(* CODESYS project UPMRACING_Driverless.project

Project tree, tasks and I/O mapping:
  Device : HY-TTC 580, TTControl, order no. n/a, version 1.2.0.0
    application Application
      libraries: Standard, * (System); lib500, 1.2.0.0 (TTControl); lib500_types, 1.2.0.0 (TTControl); lib500_syscom, 1.2.0.0 (TTControl); lib500_can2, 0.2.0.5 (TTControl); Util, * (System); Base Control Library Unsafe, 0.4.0.2 (TTControl)
      task MainTask (cyclic, interval t#10ms, priority 3, watchdog t#1000ms x 1) calls PLC_PRG
      task _ErrorCallback (externalevent, external event ErrorCallback, priority 1) calls _ErrorCB_PRG
      task _NotificationCallback (externalevent, external event NotificationCallback, priority 0) calls _NotificationCB_PRG
      program PLC_PRG [ST]
      program _NotificationCB_PRG [ST]
      program _ErrorCB_PRG [ST]
      global variables GVL
      program cl_split_byte [ST]
      CAN_Rx/
        function block CAN0_RX_Inverters [ST]
        function block CAN1_RX_V_0 [ST]
        function block CAN2_RX_V_0 [ST]
        function block CAN3_RX_V_0 [ST]
      CAN_Tx/
        function block CAN0_TX_Inverters [ST]
        function block CAN1_TX_V_0 [ST]
        function block CAN2_TX_V_0 [ST]
        function block CAN2_TX_V_1 [ST]
      UPM03/
        function block CAN_TX_V_1_4 [ST]
        function block CAN_RX_V_1_2 [ST]
        function block UPMRacing_14E_StateMachine_Antigua [ST]
      V_1/
        function block UPMRacing_14E_StateMachine [ST]
        global variables GVL_CONSTS
        function block UPMRacing_14E_StateMachine_vieja [ST]
        function block PLC_CODER_TIMER [ST]
    CANs : CANs, TTControl, order no. n/a, version 1.2.0.0
      CAN0 : CAN0, TTControl, order no. n/a, version 1.2.0.0
      CAN1 : CAN1, TTControl, order no. n/a, version 1.2.0.0
      CAN2 : CAN2, TTControl, order no. n/a, version 1.2.0.0
          settings: Baudrate = 1000
      CAN3 : CAN3, TTControl, order no. n/a, version 1.2.0.0
      CAN4 : CAN4, TTControl, order no. n/a, version 1.2.0.0
      CAN5 : CAN5, TTControl, order no. n/a, version 1.2.0.0
      CAN6 : CAN6, TTControl, order no. n/a, version 1.2.0.0
          settings: Baudrate = 250
    System : System, TTControl, order no. n/a, version 1.2.0.0
        output Application.GVL.PowerStage : BYTE  // mode
        output Application.GVL.gSafetySwitch0 : BYTE  // mode
        output Application.GVL.gSensorSupply : BYTE  // mode
        output Application.GVL.gSensorSupply : BYTE  // mode
        output Application.GVL.gSensorSupply_10 : BYTE  // mode
        output Application.GVL.Shutdown : BIT  // shutdown
        input  Application.GVL.K15 : DWORD  // Terminal_15.value
        input  Application.GVL.Wake_Up : DWORD  // WakeUp.value
        unmapped channels: error, error, mode, error, mode, error, error, error, error, error, enable_error_group_0, enable_error_group_1, enable_error_group_2, diag_status, safe_state, error, driver_init_error, UBAT, Terminal_15, WakeUp, Temperature, SSW0, SSW1, SSW2, SSUP0, SSUP1, SSUP2, status, write, boot_error, trigger_error, Powerstage, SSW0, SSW1, SSW2, SSUP0, SSUP1, SSUP2, Terminal_15, WakeUp,
          ExtShutOff0, ExtShutOff1, ExtShutOff2
      Analog_Inputs_2Mode_10V : AIN_2Mode_10V, TTControl, order no. n/a, version 1.2.0.0
        Pin 107
          <Vacío>
        Pin 131
          <Vacío>
        Pin 108
          LV_Cell_2 : IoDrvADC2Mode10, TTControl, order no. n/a, version 1.2.0.0
              input  Application.GVL.LV_Cell_2 : lib500_types.IO_ADC_STATUS  // status
              unmapped channels: reset_trigger, reset_count, reset_error
        Pin 132
          <Vacío>
        Pin 109
          LV_Cell_1 : IoDrvADC2Mode10, TTControl, order no. n/a, version 1.2.0.0
              input  Application.GVL.LV_Cell_1 : lib500_types.IO_ADC_STATUS  // status
              unmapped channels: reset_trigger, reset_count, reset_error
        Pin 133
          <Empty>
        Pin 110
          <Vacío>
        Pin 134
          <Empty>
      Analog_Inputs_2Mode_32V : AIN_2Mode_32V, TTControl, order no. n/a, version 1.2.0.0
        Pin 111
          Drive_Button : IoDrvADC2Mode32, TTControl, order no. n/a, version 1.2.0.0
              input  Application.GVL.Drive_Button : lib500_types.IO_ADC_STATUS  // status
              unmapped channels: reset_trigger, reset_count, reset_error
        Pin 135
          Shutdown_Circuit : IoDrvADC2Mode32, TTControl, order no. n/a, version 1.2.0.0
              input  Application.GVL.Shutdown_Circuit : lib500_types.IO_ADC_STATUS  // status
              unmapped channels: reset_trigger, reset_count, reset_error
        Pin 112
          Reset_Button : IoDrvADC2Mode32, TTControl, order no. n/a, version 1.2.0.0
              input  Application.GVL.Reset_Button : lib500_types.IO_ADC_STATUS  // status
              unmapped channels: reset_trigger, reset_count, reset_error
        Pin 136
          LV_Cell_6 : IoDrvADC2Mode32, TTControl, order no. n/a, version 1.2.0.0
              input  Application.GVL.LV_Cell_6 : lib500_types.IO_ADC_STATUS  // status
              unmapped channels: reset_trigger, reset_count, reset_error
        Pin 113
          LV_Cell_8 : IoDrvADC2Mode32, TTControl, order no. n/a, version 1.2.0.0
              input  Application.GVL.LV_Cell_8 : lib500_types.IO_ADC_STATUS  // status
              unmapped channels: reset_trigger, reset_count, reset_error
        Pin 137
          LV_Cell_5 : IoDrvADC2Mode32, TTControl, order no. n/a, version 1.2.0.0
              input  Application.GVL.LV_Cell_5 : lib500_types.IO_ADC_STATUS  // status
              unmapped channels: reset_trigger, reset_count, reset_error
        Pin 114
          LV_Cell_7 : IoDrvADC2Mode32, TTControl, order no. n/a, version 1.2.0.0
              input  Application.GVL.LV_Cell_7 : lib500_types.IO_ADC_STATUS  // status
              unmapped channels: reset_trigger, reset_count, reset_error
        Pin 138
          LV_Cell_4 : IoDrvADC2Mode32, TTControl, order no. n/a, version 1.2.0.0
              input  Application.GVL.LV_Cell_4 : lib500_types.IO_ADC_STATUS  // status
              unmapped channels: reset_trigger, reset_count, reset_error
      Analog_Inputs_3Mode : AIN_3Mode, TTControl, order no. n/a, version 1.2.0.0
        Pin 103
          <Vacío>
        Pin 127
          <Empty>
        Pin 104
          <Empty>
        Pin 128
          <Empty>
        Pin 105
          <Empty>
        Pin 129
          <Empty>
        Pin 106
          <Empty>
        Pin 130
          <Empty>
      Digital_Outputs_HS : HSDOUT, TTControl, order no. n/a, version 1.2.0.0
        Pin 149
          Pre_Charge : IoDrvDOSafety, TTControl, order no. n/a, version 1.2.0.0
              output Application.GVL.Pre_Charge : BIT  // output
              unmapped channels: error_code, reset_trigger, reset_count, reset_error, current, voltage_feedback
        Pin 173
          RTDS : IoDrvDOSafety, TTControl, order no. n/a, version 1.2.0.0
              output Application.GVL.RTDS_Sound : BIT  // output
              unmapped channels: error_code, reset_trigger, reset_count, reset_error, current, voltage_feedback
        Pin 152
          Brake_Light : IoDrvDOSafety, TTControl, order no. n/a, version 1.2.0.0
              output Application.GVL.Brake_Light : BIT  // output
              unmapped channels: error_code, reset_trigger, reset_count, reset_error, current, voltage_feedback
        Pin 176
          <Vacío>
        Pin 155
          <Vacío>
        Pin 179
          <Vacío>
        Pin 158
          <Vacío>
        Pin 182
          <Vacío>
      Digital_Outputs_LS : LSDOUT, TTControl, order no. n/a, version 1.2.0.0
        Pin 251
          <Empty>
        Pin 238
          <Empty>
        Pin 252
          <Empty>
        Pin 239
          <Empty>
        Pin 253
          <Empty>
        Pin 240
          <Empty>
        Pin 254
          <Empty>
        Pin 241
          <Empty>
      PVG_Outputs : PVG, TTControl, order no. n/a, version 1.2.0.0
        Pin 161
          GVL_X15_EF2_INV_1_2 : IoDrvDODiag, TTControl, order no. n/a, version 1.2.0.0
              output Application.GVL.GVL_X15_EF2_INV_1_2 : BIT  // output
              input  Application.GVL.ERROR_GVL_X15_EF2_INV_1_2 : WORD  // error_code
              unmapped channels: reset_trigger, reset_count, reset_error, current, voltage_feedback
        Pin 185
          GVL_X15_EF2_INV_3_4 : IoDrvDODiag, TTControl, order no. n/a, version 1.2.0.0
              output Application.GVL.GVL_X15_EF2_INV_3_4 : BIT  // output
              input  Application.GVL.ERROR_GVL_X15_EF2_INV_3_4 : WORD  // error_code
              unmapped channels: reset_trigger, reset_count, reset_error, current, voltage_feedback
        Pin 188
          <Empty>
        Pin 164
          <Empty>
        Pin 191
          <Empty>
        Pin 167
          <Empty>
        Pin 194
          <Vacío>
        Pin 170
          <Empty>
      PWM_Outputs : PWM, TTControl, order no. n/a, version 1.2.0.0
        Safety_switch_0 : PWM_SSW0, TTControl, order no. n/a, version 1.2.0.0
          Pin 153
            <Vacío>
          Pin 177
            <Empty>
          Pin 156
            <Empty>
          Pin 180
            <Vacío>
          Pin 159
            <Empty>
          Pin 183
            <Empty>
          Pin 186
            <Empty>
          Pin 162
            <Empty>
          Pin 189
            <Empty>
          Pin 165
            <Empty>
          Pin 192
            <Empty>
          Pin 168
            <Empty>
          Pin 195
            <Empty>
          Pin 171
            <Empty>
        Safety_switch_1 : PWM_SSW1, TTControl, order no. n/a, version 1.2.0.0
          Pin 154
            <Empty>
          Pin 178
            <Empty>
          Pin 157
            <Empty>
          Pin 181
            <Empty>
          Pin 160
            <Empty>
          Pin 184
            <Empty>
          Pin 187
            <Empty>
          Pin 163
            <Empty>
          Pin 190
            <Empty>
          Pin 166
            <Empty>
          Pin 193
            <Empty>
          Pin 169
            <Empty>
          Pin 196
            <Vacío>
          Pin 172
            <Empty>
        Safety_switch_2 : PWM_SSW2, TTControl, order no. n/a, version 1.2.0.0
          Pin 101
            <Empty>
          Pin 125
            <Empty>
          Pin 150
            <Empty>
          Pin 174
            <Empty>
          Pin 102
            <Empty>
          Pin 126
            <Empty>
          Pin 151
            <Empty>
          Pin 175
            <Empty>
      Timer_Inputs_Cur : TIN_Cur, TTControl, order no. n/a, version 1.2.0.0
        Pin 115
          <Empty>
        Pin 139
          <Empty>
        Pin 116
          <Empty>
        Pin 140
          <Empty>
        Pin 117
          <Empty>
        Pin 141
          <Empty>
      Timer_Inputs : TIN, TTControl, order no. n/a, version 1.2.0.0
        Pin 122
          <Empty>
        Pin 146
          LV_Cell_3 : IoDrvADC, TTControl, order no. n/a, version 1.2.0.0
              input  Application.GVL.LV_Cell_3 : lib500_types.IO_ADC_STATUS  // status
        Pin 123
          <Empty>
        Pin 147
          <Empty>
        Pin 124
          <Empty>
        Pin 148
          <Empty>
*)

// Device/Application/GVL
(*24-04-2019 Se añade gSensorSupply para que la ECU alimente con 5V. También se añade g delante de gK15, porque sino no funciona. *)


{attribute 'qualified_only'}
VAR_GLOBAL
	
(*SYSTEM VARIABLES*)
	(*Para que funcione la alimentacion de los sensores*)
	(* Powerstage status variable *)
	PowerStage:lib500_types.IO_POWER_STATE:=lib500_types.IO_POWER_STATE.IO_POWER_OFF;	
	(* Sensor Supply status variable 5V*)
	gSensorSupply: lib500_types.IO_POWER_STATE := lib500_types.IO_POWER_STATE.IO_POWER_OFF;  
	(* Sensor Supply status variable 10V*)    
	gSensorSupply_10 	: lib500_types.IO_POWER_STATE := lib500_types.IO_POWER_STATE.IO_POWER_OFF;   
(*VARIABLES OUT PWM*)	
	gSafetySwitch0 	: lib500_types.IO_POWER_STATE := lib500_types.IO_POWER_STATE.IO_POWER_OFF;      (* Safey Switch 0 status variable *)  
	
	Shutdown	: BOOL 	:= FALSE;		(* Flag to shutdown controller by software *)
	K15		: DWORD := 0;			(* Voltage value of K15 pin *)
	Wake_Up	: DWORD := 0;			(* Voltage value of Wake_Up pin *)
	CALL_SAFE_SHUTDOWN:BOOL:=FALSE;
		
(*SENSORES ENTRADA ANALOGICA*)
	//AccPedal_1: lib500_types.IO_ADC_STATUS; (* Voltaje del potenciómetro *)
	//AccPedal_2: lib500_types.IO_ADC_STATUS;
	//Brake_Pedal: lib500_types.IO_ADC_STATUS;
	Reset_Button: lib500_types.IO_ADC_STATUS;
	Drive_Button: lib500_types.IO_ADC_STATUS;
	(*Steering_Wheel: lib500_types.IO_ADC_STATUS;*)
	Shutdown_Circuit: lib500_types.IO_ADC_STATUS;
	(*BMS LV*)
	LV_Cell_1: lib500_types.IO_ADC_STATUS;
	LV_Cell_2: lib500_types.IO_ADC_STATUS;
	LV_Cell_3: lib500_types.IO_ADC_STATUS;
	LV_Cell_4: lib500_types.IO_ADC_STATUS;
	LV_Cell_5: lib500_types.IO_ADC_STATUS;
	LV_Cell_6: lib500_types.IO_ADC_STATUS;
	LV_Cell_7: lib500_types.IO_ADC_STATUS;
	LV_Cell_8: lib500_types.IO_ADC_STATUS;
	LV_Cell_9: lib500_types.IO_ADC_STATUS;
	
		

	

(*CAN HANDLES*)

	(* Structure for sending  CAN messages *)
	H_CAN_TX_0:tCan;
	H_CAN_TX_1:tCan; 
	H_CAN_TX_2:tCan;
	H_CAN_TX_3:tCan;
	
	(* Structure for  receiving CAN messages *)
	H_CAN_RX_0:tCan; (* INV 1 & 2 & 3 & 4 *)
	H_CAN_RX_1:tCan;  (* AIM BMS Telemtry *)
	H_CAN_RX_2:tCan;  (* LVBMS Cooling FrontSups Telemetry *)
	H_CAN_RX_3:tCan;  (* DataLogger CTMD *)
	
(*DIGITAL_OUTPUTS*)
	Brake_Light: BOOL:=FALSE;
	Pre_Charge: BOOL:=FALSE; 
	RTDS_Sound: BOOL:=FALSE;

(*PWM VARIABLES*)	
	
	
	(*RTDS_Sound: WORD:=0;*)
	
	
(*GLOBAL VARIABLES*)	
	
	Estado: LREAL:=0;
	Estado_Error: LREAL:=0;
	Info_Inverter_Error: LREAL:=0; 
	
	(*ERRORS*)
		(* ERROR_GVL_X08_INV_1_2:lib500_types.IO_ERRORTYPE:=lib500_types.IO_errortype.IO_E_OK;
		ERROR_GVL_X08_INV_3_4:lib500_types.IO_ERRORTYPE:=lib500_types.IO_errortype.IO_E_OK;
		ERROR_GVL_X15_EF_INV_1_2:lib500_types.IO_ERRORTYPE:=lib500_types.IO_errortype.IO_E_OK;
		ERROR_GVL_X15_EF_INV_3_4:lib500_types.IO_ERRORTYPE:=lib500_types.IO_errortype.IO_E_OK;
		ERROR_GVL_X140_BE1_INV_1_2:lib500_types.IO_ERRORTYPE:=lib500_types.IO_errortype.IO_E_OK;
		ERROR_GVL_X140_BE1_INV_3_4:lib500_types.IO_ERRORTYPE:=lib500_types.IO_errortype.IO_E_OK;
		ERROR_GVL_X140_BE2_INV_1_2:lib500_types.IO_ERRORTYPE:=lib500_types.IO_errortype.IO_E_OK;
		ERROR_GVL_X140_BE2_INV_3_4:lib500_types.IO_ERRORTYPE:=lib500_types.IO_errortype.IO_E_OK;
		ERROR_GVL_X15_EF2_INV_1_2:lib500_types.IO_ERRORTYPE:=lib500_types.IO_errortype.IO_E_OK;
		ERROR_GVL_X15_EF2_INV_3_4:lib500_types.IO_ERRORTYPE:=lib500_types.IO_errortype.IO_E_OK; *)
END_VAR

// Device/Application/V_1/GVL_CONSTS
VAR_GLOBAL CONSTANT
	c_UPMRacing_14_IN_NO_ACTIVE: USINT := 0;
	c_UPMRacing_14E_StateMac_IN: USINT := 1;
	c_UPMRacing_14_IN_ERROR_PRE: USINT := 2;
	c_UPMRacing_14E_StateM_IN_L: USINT := 3;
	c_UPMRacing_14E_IN_POWER_MO: USINT := 4;
	c_UPMRacing_14E_StateMa_IN_: USINT := 5;
	c_UPMRa_IN_WAITING_FOR_INV_: USINT := 6;
	c_UPMRacing_14E_StateM_IN_W: USINT := 7;
	c_UPMRacing_14E_Sta_IN_Acce: USINT := 1;
	d_UPMRacing_14E_StateMac_IN: USINT := 2;
	c_UPM_IN_BRAKE_PLAUSIBILITY: USINT := 3;
	c_UPMRac_IN_IMPLAUSIBILITY_: USINT := 4;
	c_UPMRacing_14E_Stat_IN_PRE: USINT := 5;
	c_UPMRacing_14E_StateMach_I: USINT := 6;
	c_UPMRacing_14E_IN_PRE_CHAR: USINT := 1;
	c_UPMRacing_14E_IN_PRE_CHA: USINT := 2;
	c_UPMRacing_14E_St_IN_DRIVE: USINT := 1;
	d_UPMRacing_14E_StateMach_I: USINT := 2;
	c_UPMRacing_1_IN_POWER_FRON: USINT := 3;
	c_UPMR_IN_SHUTDOWN_SEQUENCE: USINT := 4;
	c_UPMRacing_14E_S_IN_HV_STA: USINT := 1;
	d_UPMRacing_14E_S_IN_HV_STA: USINT := 2;
	e_UPMRacing_14E_S_IN_HV_STA: USINT := 3;
	f_UPMRacing_14E_S_IN_HV_STA: USINT := 4;
	g_UPMRacing_14E_S_IN_HV_STA: USINT := 5;
	h_UPMRacing_14E_S_IN_HV_STA: USINT := 6;
	c_UPMRacing_14E_IN_INIT_PRE: USINT := 7;
	c_UPMRacing_14E_St_IN_INVER: USINT := 8;
	c_UPMRacing_14E_St_IN_HV_SH: USINT := 1;
	c_UPMRacing_14E_IN_INIT_DIS: USINT := 2;
	c_UPMRacing_14_IN_INIT_DISC: USINT := 3;
	c_IN_INVERTER_CONTROLLER_SH: USINT := 4;
	c_UPMRacing_14E_St_IN_ERROR: USINT := 2;
	c_UPMRacing_14E_St_IN_RESET: USINT := 3;
	c_UPMRacing_14E_Sta_IN_DRIV: USINT := 1;
	c_UPMRacing_14_IN_POWER_REA: USINT := 3;
	c_UPMRa_IN_SHUTDOWN_SEQUENC: USINT := 4;
	c_UPMRacing_14E_Sta_IN_RESE: USINT := 3;
	e_UPMRacing_14E_StateMac_IN: USINT := 1;
	c_UPMRacing_14E_State_IN_NO: USINT := 2;
	d_UPMRacing_14E_St_IN_RESET: USINT := 3;
	c_UPMRacing_14E_Stat_IN_LIG: USINT := 1;
	c_UPMRacing_14E_State_IN_LI: USINT := 2;
	SS_OUTPUT: SINT := 3;
	SS_INITIALIZE: SINT := 0;
	SS_STEP: SINT := 1;
END_VAR

// Device/Application/PLC_PRG
PROGRAM PLC_PRG
VAR
	InitPLC: BOOL := TRUE;		(* Initialization variable *)
	Counter: DWORD := 0;		(* Local counter *)
	UPMRacing_14E_StateMachine:UPMRacing_14E_StateMachine; 
	 
	Ignition_EVCU:LREAL:=0;
	ECU_ON_K15:REAL:=0;
	
	RTDS_Sound_PLC: UINT:=0;
END_VAR

(*FUNCIONES DE INICIO SEGURO CUANDO SE ENCIENDE LA ECU*)
	IF (InitPLC = TRUE) THEN
		(*FUNCIONES PARA INICIALIZAR CAN*)
			(*CAN_TX_0*)
				CanInit(	iEnable			:= TRUE,                                (* Initialiaze CAN *) 
								iChannel		:= 0, 									(* CAN Channel 1 *)
								iCAN			:= ADR(GVL.H_CAN_TX_0), 						(* Structure for sending / receiving CAN messages *)
								iBaudrate       := 500, 								(* 500 kBit *)
								iCanIdExtended  := FALSE, 								(* Standard CAN Frame *)
								iEcuCycleTime   := T#10MS);
			(*CAN_RX_0*)
				CanInit(	iEnable			:= TRUE,                                (* Initialiaze CAN *) 
								iChannel		:= 0, 									(* CAN Channel 1 *)
								iCAN			:= ADR(GVL.H_CAN_RX_0), 						(* Structure for sending / receiving CAN messages *)
								iBaudrate       :=500, 								(* 500 kBit *)
								iCanIdExtended  := FALSE, 								(* Standard CAN Frame *)
								iEcuCycleTime   := T#10MS);
		    (*CAN_TX_1*)					
			CanInit(	iEnable			:= TRUE,                                (* Initialiaze CAN *) 
								iChannel		:= 1, 									(* CAN Channel 1 *)
								iCAN			:= ADR(GVL.H_CAN_TX_1), 						(* Structure for sending / receiving CAN messages *)
								iBaudrate       := 500, 								(* 250 kBit *)
								iCanIdExtended  := FALSE, 								(* Standard CAN Frame *)
								iEcuCycleTime   := T#10MS);
			(*CAN_RX_1*)
				CanInit(	iEnable			:= TRUE,                                (* Initialiaze CAN *) 
								iChannel		:= 1, 									(* CAN Channel 1 *)
								iCAN			:= ADR(GVL.H_CAN_RX_1), 						(* Structure for sending / receiving CAN messages *)
								iBaudrate       := 500, 								(* 250 kBit *)
								iCanIdExtended  := FALSE, 								(* Standard CAN Frame *)
								iEcuCycleTime   := T#10MS); 
							
											
			(*CAN_TX_3*)					
			CanInit(	iEnable			:= TRUE,                                (* Initialiaze CAN *) 
								iChannel		:= 3, 									(* CAN Channel 1 *)
								iCAN			:= ADR(GVL.H_CAN_TX_3), 						(* Structure for sending / receiving CAN messages *)
								iBaudrate       := 500, 								(* 500 kBit *)
								iCanIdExtended  := FALSE, 								(* Standard CAN Frame *)
								iEcuCycleTime   := T#10MS);
			(*CAN_RX_3*)
				CanInit(	iEnable			:= TRUE,                                (* Initialiaze CAN *) 
								iChannel		:= 3, 									(* CAN Channel 1 *)
								iCAN			:= ADR(GVL.H_CAN_RX_3), 						(* Structure for sending / receiving CAN messages *)
								iBaudrate       := 500, 								(* 500 kBit *)
								iCanIdExtended  := FALSE, 								(* Standard CAN Frame *)
								iEcuCycleTime   := T#10MS);

						
		    (*CAN_TX_2*)					
			CanInit(	iEnable			:= TRUE,                                (* Initialiaze CAN *) 
								iChannel		:= 2, 									(* CAN Channel 1 *)
								iCAN			:= ADR(GVL.H_CAN_TX_2), 						(* Structure for sending / receiving CAN messages *)
								iBaudrate       := 500, 								(* 500 kBit *)
								iCanIdExtended  := FALSE, 								(* Standard CAN Frame *)
								iEcuCycleTime   := T#10MS);  
			(*CAN_RX_2*)
				CanInit(	iEnable			:= TRUE,                                (* Initialiaze CAN *) 
								iChannel		:= 2, 									(* CAN Channel 1 *)
								iCAN			:= ADR(GVL.H_CAN_RX_2), 						(* Structure for sending / receiving CAN messages *)
								iBaudrate       := 500, 								(* 500 kBit *)
								iCanIdExtended  := FALSE, 								(* Standard CAN Frame *)
								iEcuCycleTime   := T#10MS); 					
	    
        (*DIGITAL_OUTPUT_POWERSTAGE*)
		GVL.PowerStage:=lib500_types.IO_POWER_STATE.IO_POWER_ON;	
		
		(*INICIALIZAR SENSOR SUPPLY*)
		//GVL.gSensorSupply  := lib500_types.IO_POWER_STATE.IO_POWER_ON;		(* Switching on Sensor Supply 0 and 1 to get 5V for Potentiometers *)
		//GVL.gSensorSupply_10  := lib500_types.IO_POWER_STATE.IO_POWER_ON_10V;		(* Switching on Sensor Supply 2 to get 10V for other Purposes *)	
		
		(*INICIALIZAR PWM OUT*)
		//GVL.gSafetySwitch0 := lib500_types.IO_POWER_STATE.IO_POWER_ON;		(* Switching on Safety Switch for PWM use *)
		(*INICILIZAR MAQUINA DE ESTADOS*)	
			
		UPMRacing_14E_StateMachine(ssMethodType:=0);
		
		
		(*FIN INICIALIZACION*)
		InitPLC := FALSE;  
END_IF

(*DIGITAL INPUTS*)
	IF (gvl.K15>3000) THEN
		ECU_ON_K15:=1;
	END_IF

(*UPMRACING14E_STATE_MACHINE RUN*)
(*Es necesario igualar las variables gobales que vienen de entradas analogicas, al mismo tiempo que se asigna valor a las globales de salida*)
	UPMRacing_14E_StateMachine(ssMethodType:=1,
		
	
			 ); 
			
			(*GVL.RTDS_Sound:=UINT_TO_WORD(65535*RTDS_Sound_PLC/DWORD_TO_UINT(GVL.K15));*)
			
	
(*SHUTDOWN ECU*)
	IF (GVL.K15< 3000) THEN			(* K15 < 3V *)
		Counter := Counter + 1;			(* Increment counter cyclically *)
		IF (Counter >= 500) THEN		
			GVL.Shutdown := TRUE;  (* Shutdown controller only after 500 cycles *)	
		END_IF
	ELSE
		Counter := 0;					(* Reset counter if K15 is HIGH again *)
	END_IF

END_PROGRAM

// Device/Application/V_1/UPMRacing_14E_StateMachine
FUNCTION_BLOCK UPMRacing_14E_StateMachine
VAR_INPUT
	ssMethodType: SINT;
	MISSION_STATUS: USINT;
	SDC: BOOL;
	FRONT_AXLE_TRQ_REQUEST: UINT;
	REAR_AXLE_TRQ_REQUEST: UINT;
	STEER_REQUEST_deg: REAL;
	DIRECTION_REQUEST: BOOL;
	Accel_longitudinal_ms2: INT;
	Accel_lateral_ms2: INT;
	Yaw_rate_degps: INT;
	HANDSHAKE: BOOL;
	ESTOP_REQUEST: BOOL;
	LAP_COUNTER: USINT;
	CONES_COUNT_ACTUAL: USINT;
	CONES_COUNT_ALL: USINT;
	VEH_SPEED_ACTUAL: USINT;
	VEH_SPEED_DEMAND: USINT;
	FRONT_MOTOR_SPEED_MAX: UINT;
	REAR_MOTOR_SPEED_MAX: UINT;
	HYD_PRESS_F_REQ_pct: USINT;
	HYD_PRESS_R_REQ_pct: USINT;
END_VAR
VAR_OUTPUT
	State_ASSI: USINT;
	Steer_actual_deg: SINT;
	AI_ESTOP_REQUEST: BOOL;
	BMS_FAULT: BOOL;
	FR_WHEEL_SPEED: UINT;
	FL_WHEEL_SPEED: UINT;
	RR_WHEEL_SPEED: UINT;
	RL_WHEEL_SPEED: UINT;
	MISSION_STATUS_FAULT: BOOL;
	GO_SIGNAL: BOOL;
	AUTONOMOUS_BRAKING_FAULT: BOOL;
	BRAKE_PLAUSIBILITY_FAULT: BOOL;
	AI_COMMS_LOST_FAULT: BOOL;
	STATUS_EBS: USINT;
	TS_SWITCH_STATUS: BOOL;
	
			//FBTX_VCU2LOG_Dynamics1 
		Speed_actual_kmh: USINT;
		Speed_target_kmh: USINT;
		Steer_target_deg: SINT;
		Brake_actual_pct: USINT;
		Brake_target_pct: USINT;
		Drive_trq_actual_pct: SINT;
		Drive_trq_target_pct: SINT;
		
//FBTX_VCU2LOG_Status 		
		State_EBS: USINT; 
		AMI_STATE: USINT;
		State_steering: BOOL;
		State_service_brake: USINT;
		
//FBTX_VCU2AI_Status
		SHUTDOWN_REQUEST: BOOL;
		STEERING_STATUS: BOOL;
		AS_STATE: USINT;
		FAULT_STATUS: BOOL;
		WARNING_STATUS: BOOL;
		WARN_BATT_TEMP_HIGH: BOOL;
		WARN_BATT_SOC_LOW: BOOL;
		HVIL_OPEN_FAULT: BOOL;
		HVIL_SHORT_FAULT: BOOL;
		EBS_FAULT: BOOL;
		OFFBOARD_CHARGER_FAULT: BOOL;
		AI_COMMS_LOST: BOOL;
		CHARGE_PROCEDURE_FAULT: BOOL;
		SHUTDOWN_CAUSE: USINT;
		
		//FBTX_VCU2AI_Drive_F
		FRONT_AXLE_TRQ: INT;
		FRONT_AXLE_TRQ_MAX: UINT;
		
		//FBTX_VCU2AI_Drive_R
		REAR_AXLE_TRQ: INT;
		REAR_AXLE_TRQ_MAX: UINT;
		
				//FBTX_VCU2AI_Steer
		ANGLE: REAL;
		ANGLE_MAX: UINT;
		ANGLE_REQUEST: INT;
		
		//FBTX_VCU2AI_Brake 	
		HYD_PRESS_F_pct: USINT;
		HYD_PRESS_R_pct: USINT;
		STATUS_BRK: USINT;
		
		//FBTX_VCU2AI_Wheel_counts
		FL_PULSE_COUNT: UINT;
		FR_PULSE_COUNT: UINT;
		RL_PULSE_COUNT: UINT;
		RR_PULSE_COUNT: UINT;
		
		//VCU_STATUS
		SM_SYS: USINT;
		SM_AS: USINT;
		R1_AI2VCU_STATUS_TIMEOUT_ERROR: BOOL;
		R1_AI2VCU_DRIVE_F_TIMEOUT_ERROR: BOOL;
		R1_AI2VCU_DRIVE_R_TIMEOUT_ERROR: BOOL;
		R1_AI2VCU_STATUS_HANDSHAKE_ERROR: BOOL;
		R1_AI2VCU_STEER_TIMEOUT_ERROR: BOOL;
		R1_AI2VCU_BRAKE_TIMEOUT_ERROR: BOOL;
		SYS_ACTION_STATE: USINT;
		WARN_BRAKE_PLAUSIBILITY: BOOL;
		WARN_KL15_UNDER_V: BOOL;
		WARN_AI_ESTOP_REQ: BOOL;
		WARN_AI_COMMS_LOST: BOOL;
		WARN_AUTO_BRAKING: BOOL;
		WARN_MISSION_STATUS: BOOL;

		
		
END_VAR
VAR
	sf_internal_predicateOutput: BOOL;
	c_is_active_c3_UPMRacing_Dr: USINT;
	is_Main: USINT;
	temporalCounter_i1: PLC_CODER_TIMER;
	AS_SWITCH_STATUS: BOOL;
	//Llamadas a las funciones de CAN (Copiar)

	
//	CAN3_RX_V_0:CAN3_RX_V_0;	
	CAN2_RX_V_0:CAN2_RX_V_0;
	CAN1_RX_V_0:CAN1_RX_V_0;
	
	CAN2_TX_V_1:CAN2_TX_V_1;
	CAN1_TX_V_0:CAN1_TX_V_0;
	
END_VAR

CAN1_RX_V_0(
		
					Accel_longitudinal_ms2_CAN => Accel_longitudinal_ms2,
					Accel_lateral_ms2_CAN => Accel_lateral_ms2,
					Yaw_rate_degps_CAN => Yaw_rate_degps,
					HANDSHAKE_CAN => HANDSHAKE,
					ESTOP_REQUEST_CAN => ESTOP_REQUEST,
					MISSION_STATUS_CAN => MISSION_STATUS,
					DIRECTION_REQUEST_CAN => DIRECTION_REQUEST,
					LAP_COUNTER_CAN => LAP_COUNTER,
					CONES_COUNT_ACTUAL_CAN => CONES_COUNT_ACTUAL,
					CONES_COUNT_ALL_CAN => CONES_COUNT_ALL,
					VEH_SPEED_ACTUAL_CAN => VEH_SPEED_ACTUAL,
					VEH_SPEED_DEMAND_CAN => VEH_SPEED_DEMAND,
					FRONT_AXLE_TRQ_REQUEST_CAN => FRONT_AXLE_TRQ_REQUEST,
					FRONT_MOTOR_SPEED_MAX_CAN => FRONT_MOTOR_SPEED_MAX,
					REAR_AXLE_TRQ_REQUEST_CAN => REAR_AXLE_TRQ_REQUEST,
					REAR_MOTOR_SPEED_MAX_CAN => REAR_MOTOR_SPEED_MAX,
					STEER_REQUEST_deg_CAN => STEER_REQUEST_deg,
					HYD_PRESS_F_REQ_pct_CAN => HYD_PRESS_F_REQ_pct,
					HYD_PRESS_R_REQ_pct_CAN => HYD_PRESS_R_REQ_pct,

);
	(* *)
		 
CAN2_RX_V_0(
					ASMS_CAN => AS_SWITCH_STATUS,
					TSMS_CAN => TS_SWITCH_STATUS,
					GO_SIGNAL_CAN => GO_SIGNAL,
					SDC_CAN => SDC,
					MISSION_STATUS_FAULT_CAN => MISSION_STATUS_FAULT,
					AUTONOMOUS_BRAKING_FAULT_CAN => AUTONOMOUS_BRAKING_FAULT,
					COMMS_LOST_REQUEST_CAN => AI_COMMS_LOST_FAULT,
					BMS_FAULT_CAN => BMS_FAULT,
					EBS_Status_CAN => STATUS_EBS,
					FL_WHEEL_SPEED_CAN => FL_WHEEL_SPEED,
					FR_WHEEL_SPEED_CAN => FR_WHEEL_SPEED,
					RL_WHEEL_SPEED_CAN => RL_WHEEL_SPEED,
					RR_WHEEL_SPEED_CAN => RR_WHEEL_SPEED,
	
		);


CASE ssMethodType OF
    0: 
        (* SystemInitialize for Chart: '<Root>/UPMRacing_Driverless_V1 ' *)
        is_Main := 0;
        temporalCounter_i1(timerAction := 1, maxTime := 0);
        c_is_active_c3_UPMRacing_Dr := 0;
    1: 
        (* Chart: '<Root>/UPMRacing_Driverless_V1 ' incorporates:
         *  Inport: '<Root>/STEER_REQUEST_deg'
         *  Outport: '<Root>/AI_COMMS_LOST_FAULT'
         *  Outport: '<Root>/AI_ESTOP_REQUEST'
         *  Outport: '<Root>/AUTONOMOUS_BRAKING_FAULT'
         *  Outport: '<Root>/BMS_FAULT'
         *  Outport: '<Root>/BRAKE_PLAUSIBILITY_FAULT'
         *  Outport: '<Root>/FL_WHEEL_SPEED'
         *  Outport: '<Root>/FR_WHEEL_SPEED'
         *  Outport: '<Root>/GO_SIGNAL'
         *  Outport: '<Root>/MISSION_STATUS_FAULT'
         *  Outport: '<Root>/RL_WHEEL_SPEED'
         *  Outport: '<Root>/RR_WHEEL_SPEED'
         *  Outport: '<Root>/STATUS_EBS'
         *  Outport: '<Root>/Steer_actual_deg'
         *  Outport: '<Root>/TS_SWITCH_STATUS' *)
        (* Gateway: UPMRacing_Driverless_V1 *)
        (* During: UPMRacing_Driverless_V1 *)

        IF c_is_active_c3_UPMRacing_Dr = 0 THEN 
            (* Entry: UPMRacing_Driverless_V1 *)
            c_is_active_c3_UPMRacing_Dr := 1;
            (* Entry Internal: UPMRacing_Driverless_V1 *)
            (* Entry Internal 'Main': '<S1>:1349' *)
            (* Transition: '<S1>:1388' *)
            is_Main := 3;
            (* Outport: '<Root>/State_ASSI' *)
            (* Entry 'AS_OFF': '<S1>:1350' *)
            (* '<S1>:1350:3' State_ASSI = 1 *)
            State_ASSI := 1;
        ELSE 
            (* During 'Main': '<S1>:1349' *)

            CASE is_Main OF
                1: 
                    (* Outport: '<Root>/State_ASSI' *)
                    State_ASSI := 3;
                    (* During 'AS_DRIVING': '<S1>:1355' *)
                    (* '<S1>:1368:1' sf_internal_predicateOutput = MISSION_STATUS == 3 &amp;... *)
                    (* '<S1>:1368:2' FR_WHEEL_SPEED<10 &amp;... *)
                    (* '<S1>:1368:3' FL_WHEEL_SPEED<10 &amp;... *)
                    (* '<S1>:1368:4' RR_WHEEL_SPEED<10 &amp;... *)
                    (* '<S1>:1368:5' RL_WHEEL_SPEED<10; *)

                    IF ((((MISSION_STATUS = 3) AND (FR_WHEEL_SPEED < 10)) AND (FL_WHEEL_SPEED < 10)) AND (RR_WHEEL_SPEED < 10)) AND (RL_WHEEL_SPEED < 10) THEN 
                        (* Transition: '<S1>:1368' *)
                        is_Main := 2;
                        (* Outport: '<Root>/State_ASSI' *)
                        (* Entry 'AS_FINISHED': '<S1>:1354' *)
                        (* '<S1>:1354:3' State_ASSI=5 *)
                        State_ASSI := 5;
                    ELSE 
                        (* '<S1>:1373:1' sf_internal_predicateOutput = SDC==0 ||... *)
                        (* '<S1>:1373:2' AS_SWITCH_STATUS == 0 ||... *)
                        (* '<S1>:1373:3' GO_SIGNAL == 0 ||... *)
                        (* '<S1>:1373:4' MISSION_STATUS_FAULT == 1 ||... *)
                        (* '<S1>:1373:5' AUTONOMOUS_BRAKING_FAULT == 1 || ...  *)
                        (* '<S1>:1373:6' BRAKE_PLAUSIBILITY_FAULT == 1 ||... *)
                        (* '<S1>:1373:7' AI_ESTOP_REQUEST == 1 ||... *)
                        (* '<S1>:1373:8' AI_COMMS_LOST_FAULT == 1 ||... *)
                        (* '<S1>:1373:9' BMS_FAULT == 1 ||... *)
                        (* '<S1>:1373:10' STATUS_EBS == 1; *)

                        IF ((((((((( NOT SDC) OR ( NOT AS_SWITCH_STATUS)) OR ( NOT GO_SIGNAL)) OR MISSION_STATUS_FAULT) OR AUTONOMOUS_BRAKING_FAULT) OR BRAKE_PLAUSIBILITY_FAULT) OR AI_ESTOP_REQUEST) OR AI_COMMS_LOST_FAULT) OR BMS_FAULT) OR (STATUS_EBS = 1) THEN 
                            (* Transition: '<S1>:1373' *)
                            is_Main := 5;
                            temporalCounter_i1(timerAction := 1, maxTime := 0);
                            (* Outport: '<Root>/State_ASSI' *)
                            (* Entry 'EMERGENCY_BRAKE': '<S1>:1353' *)
                            (* '<S1>:1353:3' State_ASSI=4 *)
                            State_ASSI := 4;
                        END_IF;

                    END_IF;

                2: 
                    (* Outport: '<Root>/State_ASSI' *)
                    State_ASSI := 5;
                    (* During 'AS_FINISHED': '<S1>:1354' *)
                    (* '<S1>:1366:1' sf_internal_predicateOutput = AS_SWITCH_STATUS == 0; *)

                    IF  NOT AS_SWITCH_STATUS THEN 
                        (* Transition: '<S1>:1366' *)
                        is_Main := 3;
                        (* Outport: '<Root>/State_ASSI' *)
                        (* Entry 'AS_OFF': '<S1>:1350' *)
                        (* '<S1>:1350:3' State_ASSI = 1 *)
                        State_ASSI := 1;
                    ELSE 
                        (* '<S1>:1367:1' sf_internal_predicateOutput = SDC==0; *)

                        IF  NOT SDC THEN 
                            (* Transition: '<S1>:1367' *)
                            is_Main := 5;
                            temporalCounter_i1(timerAction := 1, maxTime := 0);
                            (* Outport: '<Root>/State_ASSI' *)
                            (* Entry 'EMERGENCY_BRAKE': '<S1>:1353' *)
                            (* '<S1>:1353:3' State_ASSI=4 *)
                            State_ASSI := 4;
                        END_IF;

                    END_IF;

                3: 
                    (* Outport: '<Root>/State_ASSI' *)
                    State_ASSI := 1;
                    (* During 'AS_OFF': '<S1>:1350' *)
                    (* '<S1>:1356:1' sf_internal_predicateOutput = AS_SWITCH_STATUS == 1 &amp;... *)
                    (* '<S1>:1356:2' TS_SWITCH_STATUS == 1 &amp;... *)
                    (* '<S1>:1356:3' STATUS_EBS == 2 &amp;... *)
                    (* '<S1>:1356:4' MISSION_STATUS == 1; *)

                    IF ((AS_SWITCH_STATUS AND TS_SWITCH_STATUS) AND (STATUS_EBS = 2)) AND (MISSION_STATUS = 1) THEN 
                        (* Transition: '<S1>:1356' *)
                        is_Main := 4;
                        temporalCounter_i1(timerAction := 1, maxTime := 0);
                        (* Outport: '<Root>/State_ASSI' *)
                        (* Entry 'AS_READY': '<S1>:1352' *)
                        (* '<S1>:1352:3' State_ASSI=2 *)
                        State_ASSI := 2;
                    END_IF;

                4: 
                    (* Outport: '<Root>/State_ASSI' *)
                    State_ASSI := 2;
                    (* During 'AS_READY': '<S1>:1352' *)
                    (* '<S1>:1358:1' sf_internal_predicateOutput = AS_SWITCH_STATUS == 0; *)

                    IF  NOT AS_SWITCH_STATUS THEN 
                        (* Transition: '<S1>:1358' *)
                        is_Main := 3;
                        (* Outport: '<Root>/State_ASSI' *)
                        (* Entry 'AS_OFF': '<S1>:1350' *)
                        (* '<S1>:1350:3' State_ASSI = 1 *)
                        State_ASSI := 1;
                    ELSE 
                        (* '<S1>:1374:1' sf_internal_predicateOutput = SDC==0; *)

                        IF  NOT SDC THEN 
                            (* Transition: '<S1>:1374' *)
                            is_Main := 5;
                            temporalCounter_i1(timerAction := 1, maxTime := 0);
                            (* Outport: '<Root>/State_ASSI' *)
                            (* Entry 'EMERGENCY_BRAKE': '<S1>:1353' *)
                            (* '<S1>:1353:3' State_ASSI=4 *)
                            State_ASSI := 4;
                        ELSE 
                            (* '<S1>:1413:1' sf_internal_predicateOutput = after(5,sec) &amp;... *)
                            (* '<S1>:1413:2' FRONT_AXLE_TRQ_REQUEST == 0 &amp;... *)
                            (* '<S1>:1413:3' REAR_AXLE_TRQ_REQUEST  == 0 &amp;... *)
                            (* '<S1>:1413:4' STEER_REQUEST_deg  == 0 &amp;... *)
                            (* '<S1>:1413:5' Steer_actual_deg < 5  &amp;... *)
                            (* '<S1>:1413:6' DIRECTION_REQUEST == 0 &amp;... *)
                            (* '<S1>:1413:7' GO_SIGNAL == 0; *)
                            temporalCounter_i1(timerAction := 2, maxTime := 5000);
                            sf_internal_predicateOutput := temporalCounter_i1.done;

                            IF (((((sf_internal_predicateOutput AND (FRONT_AXLE_TRQ_REQUEST = 0)) AND (REAR_AXLE_TRQ_REQUEST = 0)) AND (STEER_REQUEST_deg = 0)) AND (Steer_actual_deg < 5)) AND ( NOT DIRECTION_REQUEST)) AND ( NOT GO_SIGNAL) THEN 
                                (* Transition: '<S1>:1413' *)
                                is_Main := 7;
                                (* Entry 'INTERMIDIATE': '<S1>:1412' *)
                                (* '<S1>:1412:3' State_ASSI=2 *)
                            END_IF;

                        END_IF;

                    END_IF;

                5: 
                    (* Outport: '<Root>/State_ASSI' *)
                    State_ASSI := 4;
                    (* During 'EMERGENCY_BRAKE': '<S1>:1353' *)
                    (* '<S1>:1363:1' sf_internal_predicateOutput = after(15,sec); *)
                    temporalCounter_i1(timerAction := 2, maxTime := 15000);

                    IF temporalCounter_i1.done THEN 
                        (* Transition: '<S1>:1363' *)
                        is_Main := 6;
                        (* Entry 'EMERGENCY_BRAKE_COMPLETED': '<S1>:1414' *)
                        (* '<S1>:1414:3' State_ASSI=4 *)
                    END_IF;

                6: 
                    (* Outport: '<Root>/State_ASSI' *)
                    State_ASSI := 4;
                    (* During 'EMERGENCY_BRAKE_COMPLETED': '<S1>:1414' *)
                    (* '<S1>:1416:1' sf_internal_predicateOutput = AS_SWITCH_STATUS == 0; *)

                    IF  NOT AS_SWITCH_STATUS THEN 
                        (* Transition: '<S1>:1416' *)
                        is_Main := 3;
                        (* Outport: '<Root>/State_ASSI' *)
                        (* Entry 'AS_OFF': '<S1>:1350' *)
                        (* '<S1>:1350:3' State_ASSI = 1 *)
                        State_ASSI := 1;
                    END_IF;

                ELSE
                    (* Outport: '<Root>/State_ASSI' *)
                    State_ASSI := 2;
                    (* During 'INTERMIDIATE': '<S1>:1412' *)
                    (* '<S1>:1372:1' sf_internal_predicateOutput = GO_SIGNAL == 1; *)

                    IF GO_SIGNAL THEN 
                        (* Transition: '<S1>:1372' *)
                        is_Main := 1;
                        (* Outport: '<Root>/State_ASSI' *)
                        (* Entry 'AS_DRIVING': '<S1>:1355' *)
                        (* '<S1>:1355:3' State_ASSI=3 *)
                        State_ASSI := 3;
                    ELSE 
                        (* '<S1>:1442:1' sf_internal_predicateOutput = SDC==0; *)

                        IF  NOT SDC THEN 
                            (* Transition: '<S1>:1442' *)
                            is_Main := 5;
                            temporalCounter_i1(timerAction := 1, maxTime := 0);
                            (* Outport: '<Root>/State_ASSI' *)
                            (* Entry 'EMERGENCY_BRAKE': '<S1>:1353' *)
                            (* '<S1>:1353:3' State_ASSI=4 *)
                            State_ASSI := 4;
                        ELSE 
                            (* '<S1>:1444:1' sf_internal_predicateOutput = FRONT_AXLE_TRQ_REQUEST ~= 0 ||... *)
                            (* '<S1>:1444:2' REAR_AXLE_TRQ_REQUEST  ~= 0 ||... *)
                            (* '<S1>:1444:3' STEER_REQUEST_deg  ~= 0 ||... *)
                            (* '<S1>:1444:4' Steer_actual_deg >= 5  ||... *)
                            (* '<S1>:1444:5' DIRECTION_REQUEST ~= 0; *)

                            IF ((((FRONT_AXLE_TRQ_REQUEST <> 0) OR (REAR_AXLE_TRQ_REQUEST <> 0)) OR (STEER_REQUEST_deg <> 0)) OR (Steer_actual_deg >= 5)) OR DIRECTION_REQUEST THEN 
                                (* Transition: '<S1>:1444' *)
                                is_Main := 4;
                                temporalCounter_i1(timerAction := 1, maxTime := 0);
                                (* Entry 'AS_READY': '<S1>:1352' *)
                                (* '<S1>:1352:3' State_ASSI=2 *)
                            END_IF;

                        END_IF;

                    END_IF;

            END_CASE;

        END_IF;

				AS_STATE := State_ASSI;
				ANGLE := STEER_REQUEST_deg;
				

        (* End of Chart: '<Root>/UPMRacing_Driverless_V1 ' *)
END_CASE;


CAN1_TX_V_0(
				//FBTX_VCU2LOG_Dynamics1 
		Speed_actual_kmh_CAN := Speed_actual_kmh,
		Speed_target_kmh_CAN := Speed_target_kmh,
		Steer_actual_deg_CAN := Steer_actual_deg,
		Steer_target_deg_CAN := Steer_target_deg,
		Brake_actual_pct_CAN := Brake_actual_pct, 
		Brake_target_pct_CAN := Brake_target_pct, 
		Drive_trq_actual_pct_CAN := Drive_trq_actual_pct,
		Drive_trq_target_pct_CAN := Drive_trq_target_pct, 
		
	
		//FBTX_VCU2LOG_Status 		
		State_ASSI_CAN := State_ASSI,
		State_EBS_CAN := State_EBS,  
//		AMI_STATE_CAN := AMI_STATE, 
		State_steering_CAN := State_steering, 
		State_service_brake_CAN := State_service_brake,
		
		//FBTX_VCU2AI_Status
		HANDSHAKE_CAN := HANDSHAKE,
		SHUTDOWN_REQUEST_CAN := SHUTDOWN_REQUEST,
		AS_SWITCH_STATUS_CAN := AS_SWITCH_STATUS ,
		TS_SWITCH_STATUS_CAN := TS_SWITCH_STATUS,
		GO_SIGNAL_CAN := GO_SIGNAL,
		STEERING_STATUS_CAN := STEERING_STATUS,
		AS_STATE_CAN := AS_STATE,
		FAULT_STATUS_CAN := FAULT_STATUS,
		WARNING_STATUS_CAN := WARNING_STATUS,
		WARN_BATT_TEMP_HIGH_CAN := WARN_BATT_TEMP_HIGH,
		WARN_BATT_SOC_LOW_CAN := WARN_BATT_SOC_LOW,
		AI_ESTOP_REQUEST_CAN := AI_ESTOP_REQUEST,
		HVIL_OPEN_FAULT_CAN := HVIL_OPEN_FAULT,
		HVIL_SHORT_FAULT_CAN := HVIL_SHORT_FAULT, 
		EBS_FAULT_CAN := EBS_FAULT,
		OFFBOARD_CHARGER_FAULT_CAN := OFFBOARD_CHARGER_FAULT,
		AI_COMMS_LOST_CAN := AI_COMMS_LOST,
		AUTONOMOUS_BRAKING_FAULT_CAN := AUTONOMOUS_BRAKING_FAULT,
		MISSION_STATUS_FAULT_CAN := MISSION_STATUS_FAULT, 
		CHARGE_PROCEDURE_FAULT_CAN := CHARGE_PROCEDURE_FAULT,
		BMS_FAULT_CAN := BMS_FAULT, 
		BRAKE_PLAUSIBILITY_FAULT_CAN := BRAKE_PLAUSIBILITY_FAULT, 
		SHUTDOWN_CAUSE_CAN := SHUTDOWN_CAUSE,
		
		//FBTX_VCU2AI_Drive_F
		FRONT_AXLE_TRQ_CAN := FRONT_AXLE_TRQ, 
		FRONT_AXLE_TRQ_REQUEST_CAN := FRONT_AXLE_TRQ_REQUEST,
		FRONT_AXLE_TRQ_MAX_CAN := FRONT_AXLE_TRQ_MAX, 
		
		//FBTX_VCU2AI_Drive_R
		REAR_AXLE_TRQ_CAN := REAR_AXLE_TRQ,
		REAR_AXLE_TRQ_REQUEST_CAN := REAR_AXLE_TRQ_REQUEST,
		REAR_AXLE_TRQ_MAX_CAN := REAR_AXLE_TRQ_MAX,
		
		//FBTX_VCU2AI_Steer
		ANGLE_CAN := ANGLE,
		ANGLE_MAX_CAN := ANGLE_MAX,
		ANGLE_REQUEST_CAN := ANGLE_REQUEST,
		
		//FBTX_VCU2AI_Brake 	
		HYD_PRESS_F_pct_CAN := HYD_PRESS_F_pct, 
		HYD_PRESS_F_REQ_pct_CAN := HYD_PRESS_F_REQ_pct,
		HYD_PRESS_R_pct_CAN := HYD_PRESS_R_pct,
		HYD_PRESS_R_REQ_pct_CAN := HYD_PRESS_R_REQ_pct,
		STATUS_BRK_CAN := STATUS_BRK,
		STATUS_EBS_CAN := STATUS_EBS, 
		
		//FBTX_VCU2AI_Speeds
		FL_WHEEL_SPEED_CAN := FL_WHEEL_SPEED,
    	FR_WHEEL_SPEED_CAN := FR_WHEEL_SPEED, 
	    RL_WHEEL_SPEED_CAN := RL_WHEEL_SPEED,
    	RR_WHEEL_SPEED_CAN := RR_WHEEL_SPEED, 
		
		//FBTX_VCU2AI_Wheel_counts
		FL_PULSE_COUNT_CAN := FL_PULSE_COUNT,
		FR_PULSE_COUNT_CAN := FR_PULSE_COUNT, 
		RL_PULSE_COUNT_CAN := RL_PULSE_COUNT,
		RR_PULSE_COUNT_CAN := RR_PULSE_COUNT,
		
		//VCU_STATUS
		SM_SYS_CAN := SM_SYS, 
		SM_AS_CAN := SM_AS,
		R1_AI2VCU_STATUS_TIMEOUT_ERROR_CAN := R1_AI2VCU_STATUS_TIMEOUT_ERROR,
		R1_AI2VCU_DRIVE_F_TIMEOUT_ERROR_CAN := R1_AI2VCU_DRIVE_F_TIMEOUT_ERROR,
		R1_AI2VCU_DRIVE_R_TIMEOUT_ERROR_CAN := R1_AI2VCU_DRIVE_R_TIMEOUT_ERROR, 
		R1_AI2VCU_STATUS_HANDSHAKE_ERROR_CAN := R1_AI2VCU_STATUS_HANDSHAKE_ERROR,
		R1_AI2VCU_STEER_TIMEOUT_ERROR_CAN := R1_AI2VCU_STEER_TIMEOUT_ERROR, 
		R1_AI2VCU_BRAKE_TIMEOUT_ERROR_CAN := R1_AI2VCU_BRAKE_TIMEOUT_ERROR,
		SYS_ACTION_STATE_CAN := SYS_ACTION_STATE,
		WARN_BRAKE_PLAUSIBILITY_CAN := WARN_BRAKE_PLAUSIBILITY, 
		WARN_KL15_UNDER_V_CAN := WARN_KL15_UNDER_V,
		WARN_AI_ESTOP_REQ_CAN := WARN_AI_ESTOP_REQ,
		WARN_AI_COMMS_LOST_CAN := WARN_AI_COMMS_LOST,
		WARN_AUTO_BRAKING_CAN := WARN_AUTO_BRAKING,
		WARN_MISSION_STATUS_CAN := WARN_MISSION_STATUS,
		

);
 


(*__*)

END_FUNCTION_BLOCK

// Device/Application/CAN_Rx/CAN1_RX_V_0
(* VERSION V1_0  *)

FUNCTION_BLOCK CAN1_RX_V_0
VAR_INPUT
END_VAR
VAR_OUTPUT	


			(* Analog Inputs 1 *)
		ASMS_CAN: BOOL;
		TSMS_CAN: BOOL;
		GO_SIGNAL_CAN: BOOL;
		SDC_CAN: BOOL;
		MISSION_STATUS_FAULT_CAN: BOOL;
		AUTONOMOUS_BRAKING_FAULT_CAN: BOOL;
		COMMS_LOST_REQUEST_CAN: BOOL;
		BMS_FAULT_CAN: BOOL;
		EBS_Status_CAN: USINT;
		FL_WHEEL_SPEED_CAN: USINT;
		FR_WHEEL_SPEED_CAN: USINT;
		RL_WHEEL_SPEED_CAN: USINT;
		RR_WHEEL_SPEED_CAN: USINT;
	
		

		Accel_longitudinal_ms2_CAN: INT;
		Accel_lateral_ms2_CAN:INT ;
		Yaw_rate_degps_CAN: INT;
		HANDSHAKE_CAN: BOOL; 
		ESTOP_REQUEST_CAN: BOOL; 
		MISSION_STATUS_CAN: USINT;
		DIRECTION_REQUEST_CAN: BOOL;
		LAP_COUNTER_CAN: USINT;
		CONES_COUNT_ACTUAL_CAN: USINT;
		CONES_COUNT_ALL_CAN: USINT;
		VEH_SPEED_ACTUAL_CAN: USINT;
		VEH_SPEED_DEMAND_CAN: USINT;		
		FRONT_AXLE_TRQ_REQUEST_CAN: UINT;
		FRONT_MOTOR_SPEED_MAX_CAN: UINT;
		REAR_AXLE_TRQ_REQUEST_CAN: UINT;
		REAR_MOTOR_SPEED_MAX_CAN: UINT;
		STEER_REQUEST_deg_CAN: REAL;
		HYD_PRESS_F_REQ_pct_CAN: USINT;
		HYD_PRESS_R_REQ_pct_CAN: USINT;
			
END_VAR
VAR
(*CanRx*)

		
	(* DV_Computer RX *)
		FBRX_AI2LOG_Dynamics2: CanRx;
		FBRX_AI2VCU_Status:CanRx;
		FBRX_AI2VCU_Drive_F:CanRx;		
		FBRX_AI2VCU_Drive_R:CanRx;
		FBRX_AI2VCU_Steer:CanRx;
		FBRX_AI2VCU_Brake: CanRx;
		FBRX_Analog_Inputs_1: CanRx;
		
  	
(*Time_out_Counter*)
		Counter_time_out_FBRX_AI2LOG_Dynamics2:INT:=0;
		Counter_time_out_FBRX_AI2VCU_Status:INT:=0;
		Counter_time_out_FBRX_AI2VCU_Drive_F:INT:=0;
		Counter_time_out_FBRX_AI2VCU_Drive_R:INT:=0;
		Counter_time_out_FBRX_AI2VCU_Steer:INT:=0;
		Counter_time_out_FBRX_AI2VCU_Brake:INT:=0;
		
		Counter_time_out_Analog_Inputs_1_RX:INT:=0;
		
		(*Timers*)
		Delay_Front: REAL := 0;
        Counter : USINT := 0;	
		
		
END_VAR

(*Vamos a ver si con acentos y eñes funciona esto. ó á é í *)

(* FBRX_AI2LOG_Dynamics2, ID=501*)
	    FBRX_AI2LOG_Dynamics2  (iCAN			:= ADR(GVL.H_CAN_RX_1),  				(* Structure for sending / receiving CAN messages *)
								iCanId				:= 16#501,							(* CAN Id of receiving message *) 
								iCanIdExtended		:= FALSE,  							(* Standard CAN Frame *)
								iTimeoutLimit		:= T#10MS,							(* Timeout after 500ms - Flag will be set *) 
								oByteCount			=> , 
								oData				=> , 
								oNewData			=> , 
								oCanTimeout			=> , 
								oReceiverId			=> , 
								oTooManyReceivers	=> );	
				
								
				IF FBRX_AI2LOG_Dynamics2   .oNewData THEN											(* If new CAN data is available *)
						
						Accel_longitudinal_ms2_CAN:= (FBRX_AI2LOG_Dynamics2.oData[0]+SHL(BYTE_TO_INT(FBRX_AI2VCU_Status.oData[1]),8));
						
						Accel_lateral_ms2_CAN:= (FBRX_AI2LOG_Dynamics2.oData[2]+SHL(BYTE_TO_INT(FBRX_AI2VCU_Status.oData[3]),8));
						
						Yaw_rate_degps_CAN:= (FBRX_AI2LOG_Dynamics2.oData[4]+SHL(BYTE_TO_INT(FBRX_AI2VCU_Status.oData[5]),8));
												
				ELSIF FBRX_AI2LOG_Dynamics2  .oCanTimeout THEN										(* If timeout flag is enabled switch off LedRed *)
				 
						Counter_time_out_FBRX_AI2LOG_Dynamics2:=Counter_time_out_FBRX_AI2LOG_Dynamics2+1;
				END_IF
	(*_*)		
	
(*_____________________________________________________________________*)


	(* FBRX_AI2VCU_Status, ID=510*)
	    FBRX_AI2VCU_Status  (iCAN			:= ADR(GVL.H_CAN_RX_1),  				(* Structure for sending / receiving CAN messages *)
								iCanId				:= 16#510,							(* CAN Id of receiving message *) 
								iCanIdExtended		:= FALSE,  							(* Standard CAN Frame *)
								iTimeoutLimit		:= T#10MS,							(* Timeout after 500ms - Flag will be set *) 
								oByteCount			=> , 
								oData				=> , 
								oNewData			=> , 
								oCanTimeout			=> , 
								oReceiverId			=> , 
								oTooManyReceivers	=> );	
				
								
				IF FBRX_AI2VCU_Status   .oNewData THEN											(* If new CAN data is available *)
						
						HANDSHAKE_CAN:= FBRX_AI2VCU_Status.oData[0].0;
				
						ESTOP_REQUEST_CAN:= FBRX_AI2VCU_Status.oData[1].0;
						
						MISSION_STATUS_CAN.0 := FBRX_AI2VCU_Status.oData[1].4;
						MISSION_STATUS_CAN.1 := FBRX_AI2VCU_Status.oData[1].5;
						
						DIRECTION_REQUEST_CAN := FBRX_AI2VCU_Status.oData[1].6;
						

						
						LAP_COUNTER_CAN:= INT_TO_USINT(FBRX_AI2VCU_Status.oData[3]);
						
						CONES_COUNT_ACTUAL_CAN:= INT_TO_USINT(FBRX_AI2VCU_Status.oData[4]);
						
						CONES_COUNT_ALL_CAN:= INT_TO_USINT(FBRX_AI2VCU_Status.oData[5]);
						
						VEH_SPEED_ACTUAL_CAN:= INT_TO_USINT(FBRX_AI2VCU_Status.oData[6]);
						
						VEH_SPEED_DEMAND_CAN:= INT_TO_USINT(FBRX_AI2VCU_Status.oData[7]);
						
						
						
				ELSIF FBRX_AI2VCU_Status  .oCanTimeout THEN										(* If timeout flag is enabled switch off LedRed *)
				 
						Counter_time_out_FBRX_AI2VCU_Status:=Counter_time_out_FBRX_AI2VCU_Status+1;
				END_IF
	(*_*)		
	
(*_____________________________________________________________________*)

(* FBRX_AI2VCU_Drive_F, ID=511 *)
	    FBRX_AI2VCU_Drive_F  (	iCAN			:= ADR(GVL.H_CAN_RX_1),  				(* Structure for sending / receiving CAN messages *)
								iCanId				:= 16#511,							(* CAN Id of receiving message *) 
								iCanIdExtended		:= FALSE,  							(* Standard CAN Frame *)
								iTimeoutLimit		:= T#10MS,							(* Timeout after 500ms - Flag will be set *) 
								oByteCount			=> , 
								oData				=> , 
								oNewData			=> , 
								oCanTimeout			=> , 
								oReceiverId			=> , 
								oTooManyReceivers	=> );	
				
								
				IF FBRX_AI2VCU_Drive_F  .oNewData THEN											(* If new CAN data is available *)
						
						FRONT_AXLE_TRQ_REQUEST_CAN:= (FBRX_AI2VCU_Drive_F.oData[0]+SHL(BYTE_TO_UINT(FBRX_AI2VCU_Drive_F.oData[1]),8));
						
						FRONT_MOTOR_SPEED_MAX_CAN:= (FBRX_AI2VCU_Drive_F.oData[2]+SHL(BYTE_TO_UINT(FBRX_AI2VCU_Drive_F.oData[3]),8));
							
				ELSIF FBRX_AI2VCU_Drive_F  .oCanTimeout THEN										(* If timeout flag is enabled switch off LedRed *)
				 
						Counter_time_out_FBRX_AI2VCU_Drive_F:=Counter_time_out_FBRX_AI2VCU_Drive_F+1;
				END_IF

	(*_*)		
	
(*_____________________________________________________________________*)

(* FBRX_AI2VCU_Drive_R, ID=512*)

FBRX_AI2VCU_Drive_R  (	iCAN			:= ADR(GVL.H_CAN_RX_1),  				(* Structure for sending / receiving CAN messages *)
								iCanId				:= 16#512,							(* CAN Id of receiving message *) 
								iCanIdExtended		:= FALSE,  							(* Standard CAN Frame *)
								iTimeoutLimit		:= T#10MS,							(* Timeout after 500ms - Flag will be set *) 
								oByteCount			=> , 
								oData				=> , 
								oNewData			=> , 
								oCanTimeout			=> , 
								oReceiverId			=> , 
								oTooManyReceivers	=> );	
				
								
				IF FBRX_AI2VCU_Drive_R   .oNewData THEN											(* If new CAN data is available *)
						
					REAR_AXLE_TRQ_REQUEST_CAN:= (FBRX_AI2VCU_Drive_R.oData[0]+SHL(BYTE_TO_UINT(FBRX_AI2VCU_Drive_R.oData[1]),8));
					
					REAR_MOTOR_SPEED_MAX_CAN:= (FBRX_AI2VCU_Drive_R.oData[2]+SHL(BYTE_TO_UINT(FBRX_AI2VCU_Drive_R.oData[3]),8));
					
							
				ELSIF FBRX_AI2VCU_Drive_R .oCanTimeout THEN										(* If timeout flag is enabled switch off LedRed *)
				 
						Counter_time_out_FBRX_AI2VCU_Drive_R:=Counter_time_out_FBRX_AI2VCU_Drive_R+1;
				END_IF

(*_____________________________________________________________________*)

(* FBRX_AI2VCU_Steer, ID=513*)

FBRX_AI2VCU_Steer  (	iCAN			:= ADR(GVL.H_CAN_RX_1),  				(* Structure for sending / receiving CAN messages *)
								iCanId				:= 16#513,							(* CAN Id of receiving message *) 
								iCanIdExtended		:= FALSE,  							(* Standard CAN Frame *)
								iTimeoutLimit		:= T#10MS,							(* Timeout after 500ms - Flag will be set *) 
								oByteCount			=> , 
								oData				=> , 
								oNewData			=> , 
								oCanTimeout			=> , 
								oReceiverId			=> , 
								oTooManyReceivers	=> );	
				
								
				IF FBRX_AI2VCU_Steer   .oNewData THEN											(* If new CAN data is available *)
						
					STEER_REQUEST_deg_CAN:= ((FBRX_AI2VCU_Steer.oData[0]+SHL(BYTE_TO_UINT(FBRX_AI2VCU_Steer.oData[1]),8)))/10;
										
							
				ELSIF FBRX_AI2VCU_Steer .oCanTimeout THEN										(* If timeout flag is enabled switch off LedRed *)
				 
						Counter_time_out_FBRX_AI2VCU_Steer:=Counter_time_out_FBRX_AI2VCU_Steer+1;
				END_IF

(*_____________________________________________________________________*)

(* FBRX_AI2VCU_Brake, ID=514*)

FBRX_AI2VCU_Brake  (	iCAN			:= ADR(GVL.H_CAN_RX_1),  				(* Structure for sending / receiving CAN messages *)
								iCanId				:= 16#514,							(* CAN Id of receiving message *) 
								iCanIdExtended		:= FALSE,  							(* Standard CAN Frame *)
								iTimeoutLimit		:= T#10MS,							(* Timeout after 500ms - Flag will be set *) 
								oByteCount			=> , 
								oData				=> , 
								oNewData			=> , 
								oCanTimeout			=> , 
								oReceiverId			=> , 
								oTooManyReceivers	=> );	
				
								
				IF FBRX_AI2VCU_Brake   .oNewData THEN											(* If new CAN data is available *)
						
						HYD_PRESS_F_REQ_pct_CAN:= INT_TO_USINT(FBRX_AI2VCU_Status.oData[0]);
						
						HYD_PRESS_R_REQ_pct_CAN:= INT_TO_USINT(FBRX_AI2VCU_Status.oData[1]);
										
							
				ELSIF FBRX_AI2VCU_Brake .oCanTimeout THEN										(* If timeout flag is enabled switch off LedRed *)
				 
						Counter_time_out_FBRX_AI2VCU_Brake:=Counter_time_out_FBRX_AI2VCU_Brake+1;
				END_IF
				
		
	

(*_____________________________________________________________________*)

END_FUNCTION_BLOCK

// Device/Application/CAN_Rx/CAN2_RX_V_0
(* VERSION V1_0  *)

FUNCTION_BLOCK CAN2_RX_V_0
VAR_INPUT
END_VAR
VAR_OUTPUT	
	
	(* Analog Inputs 1 *)
		ASMS_CAN: BOOL;
		TSMS_CAN: BOOL;
		GO_SIGNAL_CAN: BOOL;
		SDC_CAN: BOOL;
		MISSION_STATUS_FAULT_CAN: BOOL;
		AUTONOMOUS_BRAKING_FAULT_CAN: BOOL;
		COMMS_LOST_REQUEST_CAN: BOOL;
		BMS_FAULT_CAN: BOOL;
		EBS_Status_CAN: USINT;
		FL_WHEEL_SPEED_CAN: USINT;
		FR_WHEEL_SPEED_CAN: USINT;
		RL_WHEEL_SPEED_CAN: USINT;
		RR_WHEEL_SPEED_CAN: USINT;
	
			
END_VAR
VAR
(*CanRx*)
		
	(* Sensors RX *)
		FBRX_Analog_Inputs_1:CanRx;
			
(*Time_out_Counter*)

		Counter_time_out_Analog_Inputs_1_RX:INT:=0;
		
		(*Timers*)
		Delay_Front: REAL := 0;
        Counter : USINT := 0;

		
END_VAR


(* ESTA LÍNEA DE CAN LA USAREMOS PARA RECIBIR LAS VARIABLES QUE EN EL COCHE LE LLEGARÍAN POR ENTRADAS ANALÓGICAS *)
 

  FBRX_Analog_Inputs_1  (iCAN			:= ADR(GVL.H_CAN_RX_2),  				(* Structure for sending / receiving CAN messages *)
								iCanId				:= 16#001,							(* CAN Id of receiving message *) 
								iCanIdExtended		:= FALSE,  							(* Standard CAN Frame *)
								iTimeoutLimit		:= T#10MS,							(* Timeout after 500ms - Flag will be set *) 
								oByteCount			=> , 
								oData				=> , 
								oNewData			=> , 
								oCanTimeout			=> , 
								oReceiverId			=> , 
								oTooManyReceivers	=> );	
				
								
				IF FBRX_Analog_Inputs_1   .oNewData THEN											(* If new CAN data is available *)
					ASMS_CAN := FBRX_Analog_Inputs_1.oData[0].0;
					TSMS_CAN := FBRX_Analog_Inputs_1.oData[0].1;
					GO_SIGNAL_CAN := FBRX_Analog_Inputs_1.oData[0].2;
					SDC_CAN := FBRX_Analog_Inputs_1.oData[0].3;
					MISSION_STATUS_FAULT_CAN := FBRX_Analog_Inputs_1.oData[0].4;
					AUTONOMOUS_BRAKING_FAULT_CAN := FBRX_Analog_Inputs_1.oData[0].5;
					COMMS_LOST_REQUEST_CAN := FBRX_Analog_Inputs_1.oData[0].6;
					BMS_FAULT_CAN := FBRX_Analog_Inputs_1.oData[0].7;
					EBS_Status_CAN := INT_TO_USINT(FBRX_Analog_Inputs_1.oData[1]);
					FL_WHEEL_SPEED_CAN := INT_TO_USINT(FBRX_Analog_Inputs_1.oData[2]);
					FR_WHEEL_SPEED_CAN := INT_TO_USINT(FBRX_Analog_Inputs_1.oData[3]);
					RL_WHEEL_SPEED_CAN := INT_TO_USINT(FBRX_Analog_Inputs_1.oData[4]);
					RR_WHEEL_SPEED_CAN := INT_TO_USINT(FBRX_Analog_Inputs_1.oData[5]);
				
				ELSIF FBRX_Analog_Inputs_1  .oCanTimeout THEN										(* If timeout flag is enabled switch off LedRed *)
				 
					Counter_time_out_Analog_Inputs_1_RX:=Counter_time_out_Analog_Inputs_1_RX+1;
					
				END_IF
	

	
	
(*_____________________________________________________________________*)

END_FUNCTION_BLOCK

// Device/Application/CAN_Tx/CAN1_TX_V_0


FUNCTION_BLOCK CAN1_TX_V_0
VAR_INPUT
	
		//FBTX_VCU2LOG_Dynamics1 
		Speed_actual_kmh_CAN: USINT;
		Speed_target_kmh_CAN: USINT;
		Steer_actual_deg_CAN: SINT;
		Steer_target_deg_CAN: SINT;
		Brake_actual_pct_CAN: USINT;
		Brake_target_pct_CAN: USINT;
		Drive_trq_actual_pct_CAN: SINT;
		Drive_trq_target_pct_CAN: SINT;
		
		
		//FBTX_VCU2LOG_Status 		
		State_ASSI_CAN: USINT;
		State_EBS_CAN: USINT; 
		AMI_STATE_CAN: USINT:=2;
		State_steering_CAN: BOOL;
		State_service_brake_CAN: USINT;
		
		//FBTX_VCU2AI_Status
		HANDSHAKE_CAN: BOOL;
		SHUTDOWN_REQUEST_CAN: BOOL;
		AS_SWITCH_STATUS_CAN: BOOL;
		TS_SWITCH_STATUS_CAN: BOOL;
		GO_SIGNAL_CAN: BOOL;
		STEERING_STATUS_CAN: BOOL;
		AS_STATE_CAN: USINT;
		FAULT_STATUS_CAN: BOOL;
		WARNING_STATUS_CAN: BOOL;
		WARN_BATT_TEMP_HIGH_CAN: BOOL;
		WARN_BATT_SOC_LOW_CAN: BOOL;
		AI_ESTOP_REQUEST_CAN: BOOL;
		HVIL_OPEN_FAULT_CAN: BOOL;
		HVIL_SHORT_FAULT_CAN: BOOL;
		EBS_FAULT_CAN: BOOL;
		OFFBOARD_CHARGER_FAULT_CAN: BOOL;
		AI_COMMS_LOST_CAN: BOOL;
		AUTONOMOUS_BRAKING_FAULT_CAN: BOOL;
		MISSION_STATUS_FAULT_CAN: BOOL;
		CHARGE_PROCEDURE_FAULT_CAN: BOOL;
		BMS_FAULT_CAN: BOOL;
		BRAKE_PLAUSIBILITY_FAULT_CAN: BOOL;
		SHUTDOWN_CAUSE_CAN: USINT;
		
		//FBTX_VCU2AI_Drive_F
		FRONT_AXLE_TRQ_CAN: INT;
		FRONT_AXLE_TRQ_REQUEST_CAN: UINT;
		FRONT_AXLE_TRQ_MAX_CAN: UINT;
		
		//FBTX_VCU2AI_Drive_R
		REAR_AXLE_TRQ_CAN: INT;
		REAR_AXLE_TRQ_REQUEST_CAN: UINT;
		REAR_AXLE_TRQ_MAX_CAN: UINT;
		
		//FBTX_VCU2AI_Steer
		ANGLE_CAN: REAL;
		ANGLE_MAX_CAN: UINT;
		ANGLE_REQUEST_CAN: INT;
		
		//FBTX_VCU2AI_Brake 	
		HYD_PRESS_F_pct_CAN: USINT;
		HYD_PRESS_F_REQ_pct_CAN: USINT;
		HYD_PRESS_R_pct_CAN: USINT; 
		HYD_PRESS_R_REQ_pct_CAN: USINT;
		STATUS_BRK_CAN: USINT;
		STATUS_EBS_CAN: USINT;
		
		//FBTX_VCU2AI_Speeds
		FL_WHEEL_SPEED_CAN: UINT;
    	FR_WHEEL_SPEED_CAN: UINT;
	    RL_WHEEL_SPEED_CAN: UINT;
    	RR_WHEEL_SPEED_CAN: UINT;
		
		//FBTX_VCU2AI_Wheel_counts
		FL_PULSE_COUNT_CAN: UINT;
		FR_PULSE_COUNT_CAN: UINT;
		RL_PULSE_COUNT_CAN: UINT;
		RR_PULSE_COUNT_CAN: UINT;
		
		//VCU_STATUS
		SM_SYS_CAN: USINT;
		SM_AS_CAN: USINT;
		R1_AI2VCU_STATUS_TIMEOUT_ERROR_CAN: BOOL;
		R1_AI2VCU_DRIVE_F_TIMEOUT_ERROR_CAN: BOOL;
		R1_AI2VCU_DRIVE_R_TIMEOUT_ERROR_CAN: BOOL;
		R1_AI2VCU_STATUS_HANDSHAKE_ERROR_CAN: BOOL;
		R1_AI2VCU_STEER_TIMEOUT_ERROR_CAN: BOOL;
		R1_AI2VCU_BRAKE_TIMEOUT_ERROR_CAN: BOOL;
		SYS_ACTION_STATE_CAN: USINT;
		WARN_BRAKE_PLAUSIBILITY_CAN: BOOL;
		WARN_KL15_UNDER_V_CAN: BOOL;
		WARN_AI_ESTOP_REQ_CAN: BOOL;
		WARN_AI_COMMS_LOST_CAN: BOOL;
		WARN_AUTO_BRAKING_CAN: BOOL;
		WARN_MISSION_STATUS_CAN: BOOL;
		
END_VAR
VAR_OUTPUT
END_VAR
VAR
(*CanTX*) 

	(*Auxiliary Variable*)
		TxData: ARRAY [0..7]OF BYTE;
	
	(*AIM*)	
		FBTX_VCU2LOG_Dynamics1:CanTx;              (* Function block to send one CAN message *)
		
		FBTX_VCU2LOG_Status:CanTx;	
	
		FBTX_VCU2AI_Status:CanTx;

		FBTX_VCU2AI_Drive_F:CanTx;

		FBTX_VCU2AI_Drive_R:CanTx;

		FBTX_VCU2AI_Steer:CanTx;

		FBTX_VCU2AI_Brake:CanTx;

		FBTX_VCU2AI_Speeds:CanTx;	
		
		FBTX_VCU_Status:CanTx;
END_VAR

(*FBTX_VCU2LOG_Dynamics1, ID=500, 10ms *) 
		(*TxData=16#00*)
			TxData[0]:=16#00;
			TxData[1]:=16#00;
			TxData[2]:=16#00;
			TxData[3]:=16#00;
			TxData[4]:=16#00;
			TxData[5]:=16#00;
			TxData[6]:=16#00;
			TxData[7]:=16#00;
		(*ASIGNACION DE LA VARIABLE A LA VARIABLE A ENVIAR (TxData)*)
		TxData[0]:=USINT_TO_BYTE(Speed_actual_kmh_CAN);
		TxData[1]:=USINT_TO_BYTE(Speed_target_kmh_CAN);
		TxData[2]:=SINT_TO_BYTE(Steer_actual_deg_CAN);
		TxData[3]:=SINT_TO_BYTE(Steer_target_deg_CAN);
		TxData[4]:=USINT_TO_BYTE(Brake_actual_pct_CAN);
		TxData[5]:=USINT_TO_BYTE(Brake_target_pct_CAN);
		TxData[6]:=SINT_TO_BYTE(Drive_trq_actual_pct_CAN);
		TxData[7]:=SINT_TO_BYTE(Drive_trq_target_pct_CAN);
				
				(*ENVÍO DE TxData*)
					FBTX_VCU2LOG_Dynamics1(	iEnable				:= TRUE, 			(* Enables sending of messages *)
									iCAN				:= ADR(GVL.H_CAN_TX_1),			(* Structure for sending / receiving CAN messages *)
									iForceSend			:= FALSE,                       (* Force sending sends message immediately *)
									iTransmitRate		:= T#10MS, 						(* Cyclic transmission every 100ms *)
									iCanId				:= 16#500,						(* CAN Id for message to send *)
									iCanIdExtended		:= FALSE, 						(* Standard CAN Frame *)
									iByteCount			:= 8,							(* Number of bytes to send *)
									iData				:= TxData, 						(* Data frame *)
									oTransmitterId		=> ,
									oTooManyTransmitters=> , 
									oMsgSent			=> 
								);
(*__*)

							
(*FBTX_VCU2LOG_Status, ID=502, 10 ms *)
		(*TxData=16#00*)
			TxData[0]:=16#00;
			TxData[1]:=16#00;
			TxData[2]:=16#00;
			TxData[3]:=16#00;
			TxData[4]:=16#00;
		(*ASIGNACION DE LA VARIABLE A LA VARIABLE A ENVIAR (TxData)*)
		TxData[0]:=USINT_TO_BYTE(State_ASSI_CAN);
		TxData[1]:=USINT_TO_BYTE(State_EBS_CAN);
		TxData[2]:=USINT_TO_BYTE(AMI_STATE_CAN);
		TxData[3]:=BOOL_TO_BYTE(State_steering_CAN);
		TxData[4]:=USINT_TO_BYTE(State_service_brake_CAN);
		
									
				(*ENVÍO DE TxData*)
						FBTX_VCU2LOG_Status(	iEnable				:= TRUE, 			(* Enables sending of messages *)
									iCAN				:= ADR(GVL.H_CAN_TX_1),			(* Structure for sending / receiving CAN messages *)
									iForceSend			:= FALSE,                       (* Force sending sends message immediately *)
									iTransmitRate		:= T#10MS, 						(* Cyclic transmission every 1000ms *)
									iCanId				:= 16#502,						(* CAN Id for message to send *)
									iCanIdExtended		:= FALSE, 						(* Standard CAN Frame *)
									iByteCount			:= 5,							(* Number of bytes to send *)
									iData				:= TxData, 						(* Data frame *)
									oTransmitterId		=> ,
									oTooManyTransmitters=> , 
									oMsgSent			=> 
								);  			
(*__*)							


(*FBTX_VCU2AI_Status, ID=520, 10 ms *)
		(*TxData=16#00*)
			TxData[0]:=16#00;
			TxData[1]:=16#00;
			TxData[2]:=16#00;
			TxData[3]:=16#00;
			TxData[4]:=16#00;
			TxData[5]:=16#00;
			TxData[6]:=16#00;
			TxData[7]:=16#00;
		(*ASIGNACION DE LA VARIABLE A LA VARIABuLE A ENVIAR (TxData)*)
		TxData[0].0:=HANDSHAKE_CAN; 
		TxData[0].1:=SHUTDOWN_REQUEST_CAN; 
		TxData[0].2:=AS_SWITCH_STATUS_CAN; 
		TxData[0].3:=TS_SWITCH_STATUS_CAN; 
		TxData[0].4:=GO_SIGNAL_CAN; 
		TxData[0].5:=STEERING_STATUS_CAN; 
		
		TxData[2]:=USINT_TO_BYTE(AS_STATE_CAN);
		TxData[2].4:=AMI_STATE_CAN.0;
		TxData[2].5:=AMI_STATE_CAN.1;
		TxData[2].6:=AMI_STATE_CAN.2;
		TxData[2].7:=AMI_STATE_CAN.3;
		
		TxData[3].0:=FAULT_STATUS_CAN; 
		TxData[3].1:=WARNING_STATUS_CAN; 
		TxData[3].2:=WARN_BATT_TEMP_HIGH_CAN; 
		TxData[3].3:=WARN_BATT_SOC_LOW_CAN; 
		TxData[3].4:=AI_ESTOP_REQUEST_CAN; 
		TxData[3].5:=HVIL_OPEN_FAULT_CAN; 
		TxData[3].6:=HVIL_SHORT_FAULT_CAN; 
		TxData[3].7:=EBS_FAULT_CAN;
		
		TxData[4].0:=OFFBOARD_CHARGER_FAULT_CAN; 
		TxData[4].1:=AI_COMMS_LOST_CAN; 
		TxData[4].2:=AUTONOMOUS_BRAKING_FAULT_CAN; 
		TxData[4].3:=MISSION_STATUS_FAULT_CAN; 
		TxData[4].4:=CHARGE_PROCEDURE_FAULT_CAN; 
		TxData[4].5:=BMS_FAULT_CAN; 
		TxData[4].6:=BRAKE_PLAUSIBILITY_FAULT_CAN; 
		
		TxData[5]:=USINT_TO_BYTE(SHUTDOWN_CAUSE_CAN);
				
									
				(*ENVÍO DE TxData*)
						FBTX_VCU2AI_Status(	iEnable				:= TRUE, 			(* Enables sending of messages *)
									iCAN				:= ADR(GVL.H_CAN_TX_1),			(* Structure for sending / receiving CAN messages *)
									iForceSend			:= FALSE,                       (* Force sending sends message immediately *)
									iTransmitRate		:= T#10MS, 						(* Cyclic transmission every 1000ms *)
									iCanId				:= 16#520,						(* CAN Id for message to send *)
									iCanIdExtended		:= FALSE, 						(* Standard CAN Frame *)
									iByteCount			:= 8,							(* Number of bytes to send *)
									iData				:= TxData, 						(* Data frame *)
									oTransmitterId		=> ,
									oTooManyTransmitters=> , 
									oMsgSent			=> 
								);  			
(*__*)



(*FBTX_VCU2AI_Drive_F, ID=521, 10 ms *)
		(*TxData=16#00*)
			TxData[0]:=16#00;
			TxData[1]:=16#00;
			TxData[2]:=16#00;
			TxData[3]:=16#00;
			TxData[4]:=16#00;
			TxData[5]:=16#00;
		(*ASIGNACION DE LA VARIABLE A LA VARIABLE A ENVIAR (TxData)*)
		cl_split_dword( input := INT_TO_WORD (	DINT_TO_INT(FRONT_AXLE_TRQ_CAN + 32768)),
									byte0=>TxData[0],
									byte1=>TxData[1],
								);
		cl_split_dword( input := UINT_TO_WORD (	DINT_TO_UINT(FRONT_AXLE_TRQ_REQUEST_CAN + 32768)),
									byte0=>TxData[2],
									byte1=>TxData[3],
								);
		cl_split_dword( input := UINT_TO_WORD (	DINT_TO_UINT(FRONT_AXLE_TRQ_MAX_CAN + 32768)),
									byte0=>TxData[4],
									byte1=>TxData[5],
								);
								
				(*ENVÍO DE TxData*)
						FBTX_VCU2AI_Drive_F(	iEnable				:= TRUE, 			(* Enables sending of messages *)
									iCAN				:= ADR(GVL.H_CAN_TX_1),			(* Structure for sending / receiving CAN messages *)
									iForceSend			:= FALSE,                       (* Force sending sends message immediately *)
									iTransmitRate		:= T#10MS, 						(* Cyclic transmission every 1000ms *)
									iCanId				:= 16#521,						(* CAN Id for message to send *)
									iCanIdExtended		:= FALSE, 						(* Standard CAN Frame *)
									iByteCount			:= 6,							(* Number of bytes to send *)
									iData				:= TxData, 						(* Data frame *)
									oTransmitterId		=> ,
									oTooManyTransmitters=> , 
									oMsgSent			=> 
								);  
(*__*)



							
(*FBTX_VCU2AI_Drive_R, ID=522, 10 ms *) 
		(*TxData=16#00*)
			TxData[0]:=16#00;
			TxData[1]:=16#00;
			TxData[2]:=16#00;
			TxData[3]:=16#00;
			TxData[4]:=16#00;
			TxData[5]:=16#00;
		(*ASIGNACION DE LA VARIABLE A LA VARIABLE A ENVIAR (TxData)*)
		cl_split_dword( input := INT_TO_WORD (	DINT_TO_INT(REAR_AXLE_TRQ_CAN + 32768)),
									byte0=>TxData[0],
									byte1=>TxData[1],
								);
		cl_split_dword( input := UINT_TO_WORD (	DINT_TO_UINT(REAR_AXLE_TRQ_REQUEST_CAN + 32768)),
									byte0=>TxData[2],
									byte1=>TxData[3],
								);
		cl_split_dword( input := UINT_TO_WORD (	DINT_TO_UINT(REAR_AXLE_TRQ_MAX_CAN + 32768)),
									byte0=>TxData[4],
									byte1=>TxData[5],
								);
					
									
				(*ENVÍO DE TxData*)
						FBTX_VCU2AI_Drive_R(	iEnable				:= TRUE, 			(* Enables sending of messages *)
									iCAN				:= ADR(GVL.H_CAN_TX_1),			(* Structure for sending / receiving CAN messages *)
									iForceSend			:= FALSE,                       (* Force sending sends message immediately *)
									iTransmitRate		:= T#10MS, 						(* Cyclic transmission every 100ms *)
									iCanId				:= 16#522,						(* CAN Id for message to send *)
									iCanIdExtended		:= FALSE, 						(* Standard CAN Frame *)
									iByteCount			:= 6,							(* Number of bytes to send *)
									iData				:= TxData, 						(* Data frame *)
									oTransmitterId		=> ,
									oTooManyTransmitters=> , 
									oMsgSent			=> 
								);
(*__*)



(*FBTX_VCU2AI_Steer, ID=523, 10 ms *)
		(*TxData=16#00*)
			TxData[0]:=16#00;
			TxData[1]:=16#00;
			TxData[2]:=16#00;
			TxData[3]:=16#00;
			TxData[4]:=16#00;
			TxData[5]:=16#00;
		(*ASIGNACION DE LA VARIABLE A LA VARIABLE A ENVIAR (TxData)*)
		cl_split_dword( input := REAL_TO_WORD ((ANGLE_CAN*10)),
									byte0=>TxData[0],
									byte1=>TxData[1],
								);
								
		cl_split_dword( input := UINT_TO_WORD (	DINT_TO_UINT(ANGLE_MAX_CAN + 32768)),
									byte0=>TxData[2],
									byte1=>TxData[3],
								);
		
		cl_split_dword( input := INT_TO_WORD (	DINT_TO_INT(ANGLE_REQUEST_CAN + 32768)),
									byte0=>TxData[4],
									byte1=>TxData[5],
								);
					
									
				(*ENVÍO DE TxData*)
						FBTX_VCU2AI_Steer(	iEnable				:= TRUE, 			(* Enables sending of messages *)
									iCAN				:= ADR(GVL.H_CAN_TX_1),			(* Structure for sending / receiving CAN messages *)
									iForceSend			:= FALSE,                       (* Force sending sends message immediately *)
									iTransmitRate		:= T#10MS, 						(* Cyclic transmission every 100ms *)
									iCanId				:= 16#523,						(* CAN Id for message to send *)
									iCanIdExtended		:= FALSE, 						(* Standard CAN Frame *)
									iByteCount			:= 6,							(* Number of bytes to send *)
									iData				:= TxData, 						(* Data frame *)
									oTransmitterId		=> ,
									oTooManyTransmitters=> , 
									oMsgSent			=> 
								);
(*__*)								

	
(*FBTX_VCU2AI_Brake, ID=524, 10 ms *)
		(*TxData=16#00*)
			TxData[0]:=16#00;
			TxData[1]:=16#00;
			TxData[2]:=16#00;
			TxData[3]:=16#00;
			TxData[4]:=16#00;
			
		(*ASIGNACION DE LA VARIABLE A LA VARIABLE A ENVIAR (TxData)*)
		
	    TxData[0]:=USINT_TO_BYTE(HYD_PRESS_F_pct_CAN);
		TxData[1]:=USINT_TO_BYTE(HYD_PRESS_R_pct_CAN);
		TxData[2]:=USINT_TO_BYTE(STATUS_BRK_CAN);
		TxData[3]:=USINT_TO_BYTE(STATUS_EBS_CAN);
									
				(*ENVÍO DE TxData*)
						FBTX_VCU2AI_Brake(	iEnable				:= TRUE, 			(* Enables sending of messages *)
									iCAN				:= ADR(GVL.H_CAN_TX_1),			(* Structure for sending / receiving CAN messages *)
									iForceSend			:= FALSE,                       (* Force sending sends message immediately *)
									iTransmitRate		:= T#10MS, 						(* Cyclic transmission every 100ms *)
									iCanId				:= 16#524,						(* CAN Id for message to send *)
									iCanIdExtended		:= FALSE, 						(* Standard CAN Frame *)
									iByteCount			:= 5,							(* Number of bytes to send *)
									iData				:= TxData, 						(* Data frame *)
									oTransmitterId		=> ,
									oTooManyTransmitters=> , 
									oMsgSent			=> 
								);
								
(*__*)


(*FBTX_VCU2AI_Speeds, ID=525, 10 ms *)
		(*TxData=16#00*)
			TxData[0]:=16#00;
			TxData[1]:=16#00;
			TxData[2]:=16#00;
			TxData[3]:=16#00;
			TxData[4]:=16#00;
			TxData[5]:=16#00;
			TxData[6]:=16#00;
			TxData[7]:=16#00;
		(*ASIGNACION DE LA VARIABLE A LA VARIABLE A ENVIAR (TxData)*)
		cl_split_dword( input := UINT_TO_WORD (	DINT_TO_UINT(FL_WHEEL_SPEED_CAN + 32768)),
									byte0=>TxData[0],
									byte1=>TxData[1],
								);
		cl_split_dword( input := UINT_TO_WORD (	DINT_TO_UINT(FR_WHEEL_SPEED_CAN + 32768)),
									byte0=>TxData[2],
									byte1=>TxData[3],
								);
		cl_split_dword( input := UINT_TO_WORD (	DINT_TO_UINT(RL_WHEEL_SPEED_CAN + 32768)),
									byte0=>TxData[4],
									byte1=>TxData[5],
								);
		cl_split_dword( input := UINT_TO_WORD (	DINT_TO_UINT(RR_WHEEL_SPEED_CAN + 32768)),
									byte0=>TxData[6],
									byte1=>TxData[7],
								);
					
									
				(*ENVÍO DE TxData*)
				FBTX_VCU2AI_Speeds(	iEnable				:= TRUE, 			(* Enables sending of messages *)
									iCAN				:= ADR(GVL.H_CAN_TX_1),			(* Structure for sending / receiving CAN messages *)
									iForceSend			:= FALSE,                       (* Force sending sends message immediately *)
									iTransmitRate		:= T#10MS, 						(* Cyclic transmission every 100ms *)
									iCanId				:= 16#525,						(* CAN Id for message to send *)
									iCanIdExtended		:= FALSE, 						(* Standard CAN Frame *)
									iByteCount			:= 8,							(* Number of bytes to send *)
									iData				:= TxData, 						(* Data frame *)
									oTransmitterId		=> ,
									oTooManyTransmitters=> , 
									oMsgSent			=> 
								);
(*__*)

(*FBTX_VCU2AI_Wheel_counts, ID=526, 10 ms *)
		(*TxData=16#00*)
			TxData[0]:=16#00;
			TxData[1]:=16#00;
			TxData[2]:=16#00;
			TxData[3]:=16#00;
			TxData[4]:=16#00;
			TxData[5]:=16#00;
			TxData[6]:=16#00;
			TxData[7]:=16#00;
		(*ASIGNACION DE LA VARIABLE A LA VARIABLE A ENVIAR (TxData)*)
		cl_split_dword( input := UINT_TO_WORD (	DINT_TO_UINT(FL_PULSE_COUNT_CAN + 32768)),
									byte0=>TxData[0],
									byte1=>TxData[1],
								);
		cl_split_dword( input := UINT_TO_WORD (	DINT_TO_UINT(FR_PULSE_COUNT_CAN + 32768)),
									byte0=>TxData[2],
									byte1=>TxData[3],
								);
		cl_split_dword( input := UINT_TO_WORD (	DINT_TO_UINT(RL_PULSE_COUNT_CAN + 32768)),
									byte0=>TxData[4],
									byte1=>TxData[5],
								);
		cl_split_dword( input := UINT_TO_WORD (	DINT_TO_UINT(RR_PULSE_COUNT_CAN + 32768)),
									byte0=>TxData[6],
									byte1=>TxData[7],
								);
					
									
				(*ENVÍO DE TxData*)
				FBTX_VCU2AI_Speeds(	iEnable				:= TRUE, 			(* Enables sending of messages *)
									iCAN				:= ADR(GVL.H_CAN_TX_1),			(* Structure for sending / receiving CAN messages *)
									iForceSend			:= FALSE,                       (* Force sending sends message immediately *)
									iTransmitRate		:= T#10MS, 						(* Cyclic transmission every 100ms *)
									iCanId				:= 16#526,						(* CAN Id for message to send *)
									iCanIdExtended		:= FALSE, 						(* Standard CAN Frame *)
									iByteCount			:= 8,							(* Number of bytes to send *)
									iData				:= TxData, 						(* Data frame *)
									oTransmitterId		=> ,
									oTooManyTransmitters=> , 
									oMsgSent			=> 
								);
(*__*)

(*FBTX_VCU_Status, ID=120, 10 ms *)
		(*TxData=16#00*)
			TxData[0]:=16#00;
			TxData[1]:=16#00;
			TxData[2]:=16#00;
			TxData[3]:=16#00;
			TxData[4]:=16#00;
			TxData[5]:=16#00;
			TxData[6]:=16#00;
			TxData[7]:=16#00;
		(*ASIGNACION DE LA VARIABLE A LA VARIABLE A ENVIAR (TxData)*)
				TxData[0]:=USINT_TO_BYTE(SM_SYS_CAN);
				TxData[1]:=USINT_TO_BYTE(SM_AS_CAN);
				TxData[2].0 := R1_AI2VCU_STATUS_TIMEOUT_ERROR_CAN;
				TxData[2].1 := R1_AI2VCU_DRIVE_F_TIMEOUT_ERROR_CAN;
				TxData[2].2 := R1_AI2VCU_DRIVE_R_TIMEOUT_ERROR_CAN;
				TxData[2].3 := R1_AI2VCU_STATUS_HANDSHAKE_ERROR_CAN;
				TxData[2].4 := R1_AI2VCU_STEER_TIMEOUT_ERROR_CAN;
				TxData[2].5 := R1_AI2VCU_BRAKE_TIMEOUT_ERROR_CAN;
				TxData[3] := SYS_ACTION_STATE_CAN;
				TxData[4].0 := WARN_BRAKE_PLAUSIBILITY_CAN;
				TxData[4].1 := WARN_KL15_UNDER_V_CAN;
				TxData[4].2 := WARN_AI_ESTOP_REQ_CAN;
				TxData[4].3 := WARN_AI_COMMS_LOST_CAN;
				TxData[4].4 := WARN_AUTO_BRAKING_CAN;
				TxData[4].5 := WARN_MISSION_STATUS_CAN;

				(*ENVÍO DE TxData*)
				FBTX_VCU_Status(	iEnable				:= TRUE, 			(* Enables sending of messages *)
									iCAN				:= ADR(GVL.H_CAN_TX_1),			(* Structure for sending / receiving CAN messages *)
									iForceSend			:= FALSE,                       (* Force sending sends message immediately *)
									iTransmitRate		:= T#10MS, 						(* Cyclic transmission every 100ms *)
									iCanId				:= 16#120,						(* CAN Id for message to send *)
									iCanIdExtended		:= FALSE, 						(* Standard CAN Frame *)
									iByteCount			:= 8,							(* Number of bytes to send *)
									iData				:= TxData, 						(* Data frame *)
									oTransmitterId		=> ,
									oTooManyTransmitters=> , 
									oMsgSent			=> 
								);
(*__*)

END_FUNCTION_BLOCK

// Device/Application/V_1/PLC_CODER_TIMER
FUNCTION_BLOCK PLC_CODER_TIMER
VAR_INPUT
	timerAction: INT;
	maxTime: DINT;
END_VAR
VAR_OUTPUT
	done: BOOL;
END_VAR
VAR
	plcTimer: TON;
	plcTimerExpired: BOOL;
END_VAR


CASE timerAction OF
    1:
        (* RESET *)
        plcTimer(IN:=FALSE, PT:=T#0ms);
        plcTimerExpired := FALSE;
        done := FALSE;
    2:
        (* AFTER *)
        IF (NOT(plcTimerExpired)) THEN
            plcTimer(IN:=TRUE, PT:=DINT_TO_TIME(maxTime));
        END_IF;
        plcTimerExpired := plcTimer.Q;
        done := plcTimerExpired;
    3:
        (* BEFORE *)
        IF (NOT(plcTimerExpired)) THEN
            plcTimer(IN:=TRUE, PT:=DINT_TO_TIME(maxTime));
        END_IF;
        plcTimerExpired := plcTimer.Q;
        done := NOT(plcTimerExpired);
END_CASE;

END_FUNCTION_BLOCK

// Device/Application/CAN_Rx/CAN3_RX_V_0
(* VERSION V1_0  *)

FUNCTION_BLOCK CAN3_RX_V_0
VAR_INPUT
END_VAR
VAR_OUTPUT	
	
(*DATA_LOGGER*)
		DL_Msg_Cntr_CAN: USINT;
		DL_Status_Triggered_Current_CAN: BOOL;
		DL_Status_Triggered_Voltage_CAN: BOOL;
		DL_Status_Logging_CAN: BOOL;
		DL_Status_Ready_CAN: BOOL;
		DL_Voltage_CAN: UINT;
		DL_Current_CAN: UINT;
		
			
END_VAR
VAR
(*CanRx*)		
	
	(*DATA_LOGGER*)	
		FBRX_DATA_LOGGER:CanRx;
				
(*Time_out_Counter*)
		
	(*DATA_LOGGER*)
		Counter_time_out_DATA_LOGGER:INT:=0;	
END_VAR

(*Vamos a ver si con acentos y eñes funciona esto. ó á é í *)


(*--------------------------------------------------DATA_LOGGER--------------------------------------------------*)
	(* DATA_LOGGER, ID=430*)
		FBRX_DATA_LOGGER (	iCAN			:= ADR(GVL.H_CAN_RX_3),  				(* Structure for sending / receiving CAN messages *)
								iCanId				:= 16#430,							(* CAN Id of receiving message *) 
								iCanIdExtended		:= FALSE,  							(* Standard CAN Frame *)
								iTimeoutLimit		:= T#20MS,							(* Timeout after 500ms - Flag will be set *) 
								oByteCount			=> , 
								oData				=> , 
								oNewData			=> , 
								oCanTimeout			=> , 
								oReceiverId			=> , 
								oTooManyReceivers	=> );	
				
								
				IF FBRX_DATA_LOGGER  .oNewData THEN											(* If new CAN data is available *)
						DL_Msg_Cntr_CAN := BYTE_TO_USINT(FBRX_DATA_LOGGER.oData[0]); 
						DL_Status_Triggered_Current_CAN := FBRX_DATA_LOGGER.oData[1].3;
 						DL_Status_Triggered_Voltage_CAN := FBRX_DATA_LOGGER.oData[1].2;
						DL_Status_Logging_CAN := FBRX_DATA_LOGGER.oData[1].1;
						DL_Status_Ready_CAN := FBRX_DATA_LOGGER.oData[1].0;
						DL_Voltage_CAN := REAL_TO_UINT(16*(FBRX_DATA_LOGGER.oData[2]+SHL(BYTE_TO_UINT(FBRX_DATA_LOGGER.oData[3]),8)));
						DL_Current_CAN := REAL_TO_UINT(64*( FBRX_DATA_LOGGER.oData[4]+SHL(BYTE_TO_UINT(FBRX_DATA_LOGGER.oData[5]),8)));
						
						
						
				ELSIF FBRX_DATA_LOGGER .oCanTimeout THEN										(* If timeout flag is enabled switch off LedRed *)
				 (*Crear los errores necesarios para cuando no se leen las variable despues del time out*)
						Counter_time_out_DATA_LOGGER:=Counter_time_out_DATA_LOGGER+1;
				END_IF

(*-----------------------------------------------DATA_LOGGER--------------------------------------------------*)

END_FUNCTION_BLOCK

// Device/Application/CAN_Tx/CAN2_TX_V_1

FUNCTION_BLOCK CAN2_TX_V_1
VAR_INPUT //Crear eventualidad:para fallo de comunicación SWITCH( CAN_ERROR == 1 ) CASE PWMbomb == 100%
	// MOT_INV_1
		AMK_TempMotor1_CAN: INT;
		AMK_TempInverter1_CAN: INT;
	
	// MOT_INV_2
		AMK_TempMotor2_CAN: INT;
		AMK_TempInverter2_CAN: INT;
	
	// MOT_INV_3
		AMK_TempMotor3_CAN: INT;
		AMK_TempInverter3_CAN: INT;
	
	// MOT_INV_4
		AMK_TempMotor4_CAN: INT;
		AMK_TempInverter4_CAN: INT;
	
	// CONTROL SIGNAL
	Drive_Button_CAN: USINT;
	//AMK_bSystemReady1_CAN: BOOL;
	
		
END_VAR
VAR_OUTPUT
END_VAR
VAR
(*CanTX*)
	(*Auxiliary Variable*) 
		TxData: ARRAY [0..7] OF BYTE;
	(*MOTOR 1,2,3,4 Temperatures *)
 		Cooling_Mot_Temp: CanTx;
	(*MOTOR 1,2,3,4 Temperatures *)		
 		Cooling_Inv_Temp: CanTx;
	(*Cooling PCB Control Signals*)
		Cooling_ControlSignals: CanTx;
		
		CoolingPurge: BOOL;
		CoolingDrive: BOOL;

END_VAR

(*--------------------------------------------------Sensors TX-------------------------------------------------------------*)

(*Cooling PCB ID = 001	(CONTROL)	*)		
(* Inicialización de TxData 16#00 (Hexadecimal) *)
	TxData[0]:= 16#00;
	TxData[1]:= 16#00;
	TxData[2]:= 16#00;
	TxData[3]:= 16#00;
	TxData[4]:= 16#00;
	TxData[5]:= 16#00;
	TxData[6]:= 16#00;
	TxData[7]:= 16#00;			
	
(* Asignación de las variables a enviar a TxData *)

(* Ponemos a true o false las variables de control en funcion de si Drive esta dado e Inv encendidos 
 para la máquina de estados de cooling*)
 //Si recibimos Temp de Inverters significa que está pulsado el boton y queremos purgar
	IF (AMK_TempMotor1_CAN > 0 )AND (Drive_Button_CAN=10) THEN  
		CoolingPurge := TRUE;		
	ELSE 
		CoolingPurge := FALSE;
	END_IF
	//CoolingPurge := FALSE;
	
	(*IF (AMK_bSystemReady1_CAN = TRUE ) THEN  
		CoolingDrive := TRUE;		
	ELSE 
		CoolingDrive := FALSE;
	END_IF *)
	IF (Drive_Button_CAN > 10 ) THEN  
		CoolingDrive := TRUE;		
	ELSE 
		CoolingDrive := FALSE;
	END_IF
	
	TxData [0].0 := CoolingDrive;
	TxData [0].1 := CoolingPurge;
	
	(*ENVÍO DEL MENSAJE TxData en Cooling_ControlSignals*)
				Cooling_ControlSignals(	iEnable				:= TRUE, 							(* Enables sending of messages *)
								iCAN				:= ADR(GVL.H_CAN_TX_2),					(* Structure for sending / receiving CAN messages *)
								iForceSend			:= FALSE,                           (* Force sending sends message immediately *)
								iTransmitRate		:= T#100MS, 						(* Cyclic transmission every 100ms *)
								iCanId				:= 16#001,							(* CAN Id for message to send *)
								iCanIdExtended		:= FALSE, 							(* Standard CAN Frame *)
								iByteCount			:= 8,								(* Number of bytes to send *)
								iData				:= TxData, 							(* Data frame *)
								oTransmitterId		=> ,
								oTooManyTransmitters=> , 
								oMsgSent			=> 
								);
								
(* Cooling PCB ID = 002 (MOTORS) *)
(* Inicialización de TxData 16#00 (Hexadecimal) *)
	TxData[0]:= 16#00;
	TxData[1]:= 16#00;
	TxData[2]:= 16#00;
	TxData[3]:= 16#00;
	TxData[4]:= 16#00;
	TxData[5]:= 16#00;
	TxData[6]:= 16#00;
	TxData[7]:= 16#00;
	
(* Asignación de las variables a enviar a TxData *)
	cl_split_word( input := INT_TO_WORD (AMK_TempMotor1_CAN), 
		byte0=>TxData[0],
		byte1=>TxData[1],
	);
	cl_split_word( input := INT_TO_WORD (AMK_TempMotor2_CAN), 
		byte0=>TxData[2],
		byte1=>TxData[3],
	);
	cl_split_word( input := INT_TO_WORD (AMK_TempMotor3_CAN), 
		byte0=>TxData[4],
		byte1=>TxData[5],
	);
	cl_split_word( input := INT_TO_WORD (AMK_TempMotor4_CAN), 
		byte0=>TxData[6],
		byte1=>TxData[7],
	);

(*ENVÍO DEL MENSAJE TxData en Cooling_Mot_Temp*)
				Cooling_Mot_Temp(	iEnable				:= TRUE, 							(* Enables sending of messages *)
								iCAN				:= ADR(GVL.H_CAN_TX_2),					(* Structure for sending / receiving CAN messages *)
								iForceSend			:= FALSE,                           (* Force sending sends message immediately *)
								iTransmitRate		:= T#100MS, 						(* Cyclic transmission every 100ms *)
								iCanId				:= 16#002,							(* CAN Id for message to send *)
								iCanIdExtended		:= FALSE, 							(* Standard CAN Frame *)
								iByteCount			:= 8,								(* Number of bytes to send *)
								iData				:= TxData, 							(* Data frame *)
								oTransmitterId		=> ,
								oTooManyTransmitters=> , 
								oMsgSent			=> 
								);
								
								
(*Cooling PCB ID = 002	(INVERTERS)	*)		
(* Inicialización de TxData 16#00 (Hexadecimal) *)
	TxData[0]:= 16#00;
	TxData[1]:= 16#00;
	TxData[2]:= 16#00;
	TxData[3]:= 16#00;
	TxData[4]:= 16#00;
	TxData[5]:= 16#00;
	TxData[6]:= 16#00;
	TxData[7]:= 16#00;			
	
(* Asignación de las variables a enviar a TxData *)
	cl_split_word( input := INT_TO_WORD (AMK_TempInverter1_CAN), 
		byte0=>TxData[0],
		byte1=>TxData[1],
	);
	cl_split_word( input := INT_TO_WORD (AMK_TempInverter2_CAN), 
		byte0=>TxData[2],
		byte1=>TxData[3],
	);
	cl_split_word( input := INT_TO_WORD (AMK_TempInverter3_CAN), 
		byte0=>TxData[4],
		byte1=>TxData[5],
	);
	cl_split_word( input := INT_TO_WORD (AMK_TempInverter4_CAN), 
		byte0=>TxData[6],
		byte1=>TxData[7],
	);								
	(*ENVÍO DEL MENSAJE TxData en Cooling_Inv_Temp*)
				Cooling_Inv_Temp(	iEnable				:= TRUE, 							(* Enables sending of messages *)
								iCAN				:= ADR(GVL.H_CAN_TX_2),					(* Structure for sending / receiving CAN messages *)
								iForceSend			:= FALSE,                           (* Force sending sends message immediately *)
								iTransmitRate		:= T#100MS, 						(* Cyclic transmission every 100ms *)
								iCanId				:= 16#003,							(* CAN Id for message to send *)
								iCanIdExtended		:= FALSE, 							(* Standard CAN Frame *)
								iByteCount			:= 8,								(* Number of bytes to send *)
								iData				:= TxData, 							(* Data frame *)
								oTransmitterId		=> ,
								oTooManyTransmitters=> , 
								oMsgSent			=> 
								);
	
(*__*)


(*-----------------------------------------------FIN Sensors TX--------------------------------------------------------------*)

END_FUNCTION_BLOCK

// Device/Application/_ErrorCB_PRG
PROGRAM _ErrorCB_PRG
VAR
	diag_state : lib500_types.DIAG_STATETYPE := lib500_types.DIAG_STATETYPE.DIAG_STATE_DISABLED;
	watchdog_state : lib500_types.DIAG_WD_STATETYPE := lib500_types.DIAG_WD_STATETYPE.DIAG_WD_STATE_UNKNOWN;
	error : lib500_types.DIAG_ERRORCODE := (error_code := lib500_types.DIAG_ERRORTYPE.DIAG_E_NOERROR, 
                                            device_num := lib500_types.DIAG_DEVICETYPE.DIAG_DEV_NONE,
                                            faulty_value := 0);
	return_code : lib500_types.IO_ERRORTYPE := lib500_types.IO_ERRORTYPE.IO_E_UNKNOWN;
	
	reaction : lib500_types.DIAG_REACTION := lib500_types.DIAG_REACTION.DIAG_ERR_SAFESTATE;
	
	call_count : UDINT := 0;
END_VAR

(* get the reason for the error callback *)
return_code := lib500.DIAG_CDS_GetErrorReason(ADR(diag_state), 
                                              ADR(watchdog_state),
                                              ADR(error));

(* custom handler code can be placed here *)

(* the choices for the reactions are:
   -> lib500_types.DIAG_REACTION.DIAG_ERR_NOACTION
   -> lib500_types.DIAG_REACTION.DIAG_ERR_SAFESTATE
   -> lib500_types.DIAG_REACTION.DIAG_ERR_DISABLE_SSW0
   -> lib500_types.DIAG_REACTION.DIAG_ERR_DISABLE_SSW1
   -> lib500_types.DIAG_REACTION.DIAG_ERR_DISABLE_SSW2
   -> lib500_types.DIAG_REACTION.DIAG_ERR_DISABLE_HS00
   -> lib500_types.DIAG_REACTION.DIAG_ERR_DISABLE_HS01
   -> lib500_types.DIAG_REACTION.DIAG_ERR_DISABLE_HS02
   -> lib500_types.DIAG_REACTION.DIAG_ERR_DISABLE_HS03
   -> lib500_types.DIAG_REACTION.DIAG_ERR_DISABLE_HS04
   -> lib500_types.DIAG_REACTION.DIAG_ERR_DISABLE_HS05
   -> lib500_types.DIAG_REACTION.DIAG_ERR_DISABLE_HS06
   -> lib500_types.DIAG_REACTION.DIAG_ERR_DISABLE_HS07
   
   it's also possible to combine (binary-or) reactions, like:
   -> lib500_types.DIAG_REACTION.DIAG_ERR_DISABLE_SSW0 OR 
      lib500_types.DIAG_REACTION.DIAG_ERR_DISABLE_SSW1
*)

(* pass the error reaction to the DIAG system *)
lib500.DIAG_CDS_SetErrorReaction(reaction);

(* increment call count *)
call_count := call_count + 1;

END_PROGRAM

// Device/Application/_NotificationCB_PRG
PROGRAM _NotificationCB_PRG
VAR
	diag_state : lib500_types.DIAG_STATETYPE := lib500_types.DIAG_STATETYPE.DIAG_STATE_DISABLED;
	watchdog_state : lib500_types.DIAG_WD_STATETYPE := lib500_types.DIAG_WD_STATETYPE.DIAG_WD_STATE_UNKNOWN;
	error : lib500_types.DIAG_ERRORCODE := (error_code := lib500_types.DIAG_ERRORTYPE.DIAG_E_NOERROR, 
                                            device_num := lib500_types.DIAG_DEVICETYPE.DIAG_DEV_NONE,
                                            faulty_value := 0);
	return_code : lib500_types.IO_ERRORTYPE := lib500_types.IO_ERRORTYPE.IO_E_UNKNOWN;
	
	call_count : UDINT := 0;
END_VAR

(* get the reason for the notification callback *)
return_code := lib500.DIAG_CDS_GetNotificationReason(ADR(diag_state), 
                                                     ADR(watchdog_state),
                                                     ADR(error));

(* custom handler code can be placed here *)

(* increment call count *)
call_count := call_count + 1;

END_PROGRAM

// Device/Application/cl_split_byte
PROGRAM cl_split_byte
VAR_INPUT
	input	        : WORD;		(* word to be split *)
END_VAR
VAR_OUTPUT
	bit0	: BOOL;		(* value of bit 0 *)
	bit1	: BOOL;		(* value of bit 1 *)
	bit2	: BOOL;		(* value of bit 2 *)
	bit3	: BOOL;		(* value of bit 3 *)
END_VAR
VAR
	input_local:BYTE;
END_VAR

input_local:= WORD_TO_BYTE (input);
bit3 := input_local.3;
bit2 := input_local.2;
bit1 := input_local.1;
bit0 := input_local.0;

END_PROGRAM

// Device/Application/CAN_Tx/CAN0_TX_Inverters

(* 2019/06/25	VERSION V1_1 : Introduccion de la linea de CAN de la AIM para enviar datos de estados de la EVCU *)

FUNCTION_BLOCK CAN0_TX_Inverters
VAR_INPUT
	(*AMK_Setpoints_1_INV1, ID=184*)
		AMK_bInverterOn1_CAN: BOOL;
		AMK_bDcOn1_CAN: BOOL;
		AMK_bEnable1_CAN: BOOL;
		AMK_bErrorReset1_CAN: BOOL;
		AMK_TargetVelocity1_CAN: INT;
		AMK_TorqueLimitPositiv1_CAN: INT;
		AMK_TorqueLimitNegativ1_CAN: INT;
		
			(*AMK_Setpoints_1_INV2, ID=185*)
		AMK_bInverterOn2_CAN: BOOL;
		AMK_bDcOn2_CAN: BOOL;
		AMK_bEnable2_CAN: BOOL;
		AMK_bErrorReset2_CAN: BOOL;
		AMK_TargetVelocity2_CAN: INT;
		AMK_TorqueLimitPositiv2_CAN: INT;
		AMK_TorqueLimitNegativ2_CAN: INT;
		
		AMK_bInverterOn3_CAN: BOOL;
		AMK_bDcOn3_CAN: BOOL;
		AMK_bEnable3_CAN: BOOL;
		AMK_bErrorReset3_CAN: BOOL;
		AMK_TargetVelocity3_CAN: INT;
		AMK_TorqueLimitPositiv3_CAN: INT;
		AMK_TorqueLimitNegativ3_CAN: INT;
		
		AMK_bInverterOn4_CAN: BOOL;
		AMK_bDcOn4_CAN: BOOL;
		AMK_bEnable4_CAN: BOOL;
		AMK_bErrorReset4_CAN: BOOL;
		AMK_TargetVelocity4_CAN: INT;
		AMK_TorqueLimitPositiv4_CAN: INT;
		AMK_TorqueLimitNegativ4_CAN: INT;
	(*	
		
		Brake_Light_CAN: BOOL;
		Pre_Charge_CAN: BOOL;
		Estado_CAN: LREAL;
		Info_Inverter_Error_CAN: UINT;
		Estado_Error_CAN: LREAL;
		
		AIM_TempMotor1_CAN: INT;
		AIM_TempInverter1_CAN: INT; 
		AIM_TempMotor2_CAN: INT;
		AIM_TempInverter2_CAN: INT;
		AIM_TempMotor3_CAN: INT;
		AIM_TempInverter3_CAN: INT;
		AIM_TempMotor4_CAN: INT;
		AIM_TempInverter4_CAN: INT;	
		*)
END_VAR
VAR_OUTPUT
END_VAR
VAR
(*CanTX*)
	(*Auxiliary Variable*)
		TxData: ARRAY [0..7]OF BYTE;
	(*INVERTER_1*)
		FBTX_AMK_Setpoints_1_INV1:CanTx;              (* Function block to send one CAN message *)
	(*INVERTER_2*)
		FBTX_AMK_Setpoints_1_INV2:CanTx;              (* Function block to send one CAN message *)
	(*INVERTER_3*)
		FBTX_AMK_Setpoints_1_INV3:CanTx;              (* Function block to send one CAN message *)
	(*INVERTER_4*)
		FBTX_AMK_Setpoints_1_INV4:CanTx;              (* Function block to send one CAN message *)
(*	(*AIM*)	
		FBTX_AIM_1:CanTx;              (* Function block to send one CAN message *)
		
		FBTX_AIM_2:CanTx;	
	
		FBTX_AIM_3:CanTx;		*)

END_VAR

(*--------------------------------------------------INVERTER_1_TX--------------------------------------------------*)
	(*AMK_Setpoints_1_INV1, ID=184*)
		(*TxData=16#00*)
			TxData[0]:=16#00;
			TxData[1]:=16#00;
			TxData[2]:=16#00;
			TxData[3]:=16#00;
			TxData[4]:=16#00;
			TxData[5]:=16#00;
			TxData[6]:=16#00;
			TxData[7]:=16#00;
		(*ASIGNACION DE LA VARIABLE A LA VARIABLE A ENVIAR (TxData)*)
					TxData[1].0:=AMK_bInverterOn1_CAN;
					TxData[1].1:=AMK_bDcOn1_CAN;
					TxData[1].2:=AMK_bEnable1_CAN;
					TxData[1].3:=AMK_bErrorReset1_CAN; 
					cl_split_dword( input := REAL_TO_WORD (AMK_TargetVelocity1_CAN),
									byte0=>TxData[2],
									byte1=>TxData[3],
								);	
					cl_split_dword( input := REAL_TO_WORD (AMK_TorqueLimitPositiv1_CAN),
									byte0=>TxData[4],
									byte1=>TxData[5],
								);
					cl_split_dword( input := REAL_TO_WORD (AMK_TorqueLimitNegativ1_CAN),
									byte0=>TxData[6],
									byte1=>TxData[7],
								);										
				(*ENVÍO DE TxData*)
					FBTX_AMK_Setpoints_1_INV1(	iEnable				:= TRUE, 			(* Enables sending of messages *)
									iCAN				:= ADR(GVL.H_CAN_TX_0),			(* Structure for sending / receiving CAN messages *)
									iForceSend			:= FALSE,                       (* Force sending sends message immediately *)
									iTransmitRate		:= T#10MS, 						(* Cyclic transmission every 100ms *)
									iCanId				:= 16#184,						(* CAN Id for message to send *)
									iCanIdExtended		:= FALSE, 						(* Standard CAN Frame *)
									iByteCount			:= 8,							(* Number of bytes to send *)
									iData				:= TxData, 						(* Data frame *)
									oTransmitterId		=> ,
									oTooManyTransmitters=> , 
									oMsgSent			=> 
								);
(*-----------------------------------------------FIN_INVERTER_1_TX--------------------------------------------------*)


(*--------------------------------------------------INVERTER_2_TX--------------------------------------------------*)
	(*AMK_Setpoints_1_INV2, ID=185*)
		(*TxData=16#00*)
			TxData[0]:=16#00;
			TxData[1]:=16#00;
			TxData[2]:=16#00;
			TxData[3]:=16#00;
			TxData[4]:=16#00;
			TxData[5]:=16#00;
			TxData[6]:=16#00;
			TxData[7]:=16#00;
		(*ASIGNACION DE LA VARIABLE A LA VARIABLE A ENVIAR (TxData)*)
					TxData[1].0:=AMK_bInverterOn2_CAN;
					TxData[1].1:=AMK_bDcOn2_CAN;
					TxData[1].2:=AMK_bEnable2_CAN;
					TxData[1].3:=AMK_bErrorReset2_CAN;
					cl_split_dword( input := REAL_TO_WORD (AMK_TargetVelocity2_CAN),
									byte0=>TxData[2],
									byte1=>TxData[3],
								);	
					cl_split_dword( input := REAL_TO_WORD (AMK_TorqueLimitPositiv2_CAN),
									byte0=>TxData[4],
									byte1=>TxData[5],
								);
					cl_split_dword( input := REAL_TO_WORD (AMK_TorqueLimitNegativ2_CAN),
									byte0=>TxData[6],
									byte1=>TxData[7],
								);											
				(*ENVÍO DE TxData*)
					FBTX_AMK_Setpoints_1_INV2(	iEnable				:= TRUE, 							(* Enables sending of messages *)
									iCAN				:= ADR(GVL.H_CAN_TX_0),					(* Structure for sending / receiving CAN messages *)
									iForceSend			:= FALSE,                           (* Force sending sends message immediately *)
									iTransmitRate		:= T#10MS, 						(* Cyclic transmission every 100ms *)
									iCanId				:= 16#185,							(* CAN Id for message to send *)
									iCanIdExtended		:= FALSE, 							(* Standard CAN Frame *)
									iByteCount			:= 8,								(* Number of bytes to send *)
									iData				:= TxData, 							(* Data frame *)
									oTransmitterId		=> ,
									oTooManyTransmitters=> , 
									oMsgSent			=> 
								);
(*-----------------------------------------------FIN_INVERTER_2_TX--------------------------------------------------*)


(*--------------------------------------------------INVERTER_3_TX--------------------------------------------------*)
	(*AMK_Setpoints_1_INV3, ID=188*)
		(*TxData=16#00*)
			TxData[0]:=16#00;
			TxData[1]:=16#00;
			TxData[2]:=16#00;
			TxData[3]:=16#00;
			TxData[4]:=16#00;
			TxData[5]:=16#00;
			TxData[6]:=16#00;
			TxData[7]:=16#00;
		(*ASIGNACION DE LA VARIABLE A LA VARIABLE A ENVIAR (TxData)*)
					TxData[1].0:=AMK_bInverterOn3_CAN;
					TxData[1].1:=AMK_bDcOn3_CAN;
					TxData[1].2:=AMK_bEnable3_CAN;
					TxData[1].3:=AMK_bErrorReset3_CAN;
					cl_split_dword( input := REAL_TO_WORD (AMK_TargetVelocity3_CAN),
									byte0=>TxData[2],
									byte1=>TxData[3],
								);	
					cl_split_dword( input := REAL_TO_WORD (AMK_TorqueLimitPositiv3_CAN),
									byte0=>TxData[4],
									byte1=>TxData[5],
								);
					cl_split_dword( input := REAL_TO_WORD (AMK_TorqueLimitNegativ3_CAN),
									byte0=>TxData[6],
									byte1=>TxData[7],
								);											
				(*ENVÍO DE TxData*)
					FBTX_AMK_Setpoints_1_INV3(	iEnable				:= TRUE, 							(* Enables sending of messages *)
									iCAN				:= ADR(GVL.H_CAN_TX_0),					(* Structure for sending / receiving CAN messages *)
									iForceSend			:= FALSE,                           (* Force sending sends message immediately *)
									iTransmitRate		:= T#10MS, 						(* Cyclic transmission every 100ms *)
									iCanId				:= 16#188,							(* CAN Id for message to send *)
									iCanIdExtended		:= FALSE, 							(* Standard CAN Frame *)
									iByteCount			:= 8,								(* Number of bytes to send *)
									iData				:= TxData, 							(* Data frame *)
									oTransmitterId		=> ,
									oTooManyTransmitters=> , 
									oMsgSent			=> 
								);
(*-----------------------------------------------FIN_INVERTER_3_TX--------------------------------------------------*)



(*--------------------------------------------------INVERTER_4_TX--------------------------------------------------*)
	(*AMK_Setpoints_1_INV4, ID=189*)
		(*TxData=16#00*)
			TxData[0]:=16#00;
			TxData[1]:=16#00;
			TxData[2]:=16#00;
			TxData[3]:=16#00;
			TxData[4]:=16#00;
			TxData[5]:=16#00;
			TxData[6]:=16#00;
			TxData[7]:=16#00;
		(*ASIGNACION DE LA VARIABLE A LA VARIABLE A ENVIAR (TxData)*)
					TxData[1].0:=AMK_bInverterOn4_CAN;
					TxData[1].1:=AMK_bDcOn4_CAN;
					TxData[1].2:=AMK_bEnable4_CAN;
					TxData[1].3:=AMK_bErrorReset4_CAN;
					cl_split_dword( input := REAL_TO_WORD (AMK_TargetVelocity4_CAN),
									byte0=>TxData[2],
									byte1=>TxData[3],
								);	
					cl_split_dword( input := REAL_TO_WORD (AMK_TorqueLimitPositiv4_CAN),
									byte0=>TxData[4],
									byte1=>TxData[5],
								);
					cl_split_dword( input := REAL_TO_WORD (AMK_TorqueLimitNegativ4_CAN),
									byte0=>TxData[6],
									byte1=>TxData[7],
								);											
				(*ENVÍO DE TxData*)
					FBTX_AMK_Setpoints_1_INV4(	iEnable				:= TRUE, 							(* Enables sending of messages *)
									iCAN				:= ADR(GVL.H_CAN_TX_0),					(* Structure for sending / receiving CAN messages *)
									iForceSend			:= FALSE,                           (* Force sending sends message immediately *)
									iTransmitRate		:= T#10MS, 						(* Cyclic transmission every 100ms *)
									iCanId				:= 16#189,							(* CAN Id for message to send *)
									iCanIdExtended		:= FALSE, 							(* Standard CAN Frame *)
									iByteCount			:= 8,								(* Number of bytes to send *)
									iData				:= TxData, 							(* Data frame *)
									oTransmitterId		=> ,
									oTooManyTransmitters=> , 
									oMsgSent			=> 
								);
(*-----------------------------------------------FIN_INVERTER_4_TX--------------------------------------------------*) 
(*
(*--------------------------------------------------AIM-------------------------------------------------------------*)
(*Info_To_AIM, ID=180*)
		(*TxData=16#00*)
			TxData[0]:=16#00;
			TxData[1]:=16#00;
			TxData[2]:=16#00;
			TxData[3]:=16#00;
			TxData[4]:=16#00;
			TxData[5]:=16#00;
			TxData[6]:=16#00;
			TxData[7]:=16#00;
		(*ASIGNACION DE LA VARIABLE A LA VARIABLE A ENVIAR (TxData)*)
		cl_split_dword( input := LREAL_TO_WORD (Estado_CAN),
									byte0=>TxData[0],
									byte1=>TxData[1],
								);
		cl_split_dword( input := LREAL_TO_WORD (Estado_Error_CAN),
									byte0=>TxData[2],
									byte1=>TxData[3],
								);
		cl_split_dword( input := UINT_TO_WORD (Info_Inverter_Error_CAN),
									byte0=>TxData[4],
									byte1=>TxData[5],
								);
					TxData[6].0:=Brake_Light_CAN;
					TxData[6].1:=Pre_Charge_CAN;
									
				(*ENVÍO DE TxData*)
					FBTX_AIM_1(	iEnable				:= TRUE, 			(* Enables sending of messages *)
									iCAN				:= ADR(GVL.H_CAN_TX_6),			(* Structure for sending / receiving CAN messages *)
									iForceSend			:= FALSE,                       (* Force sending sends message immediately *)
									iTransmitRate		:= T#10MS, 						(* Cyclic transmission every 100ms *)
									iCanId				:= 16#180,						(* CAN Id for message to send *)
									iCanIdExtended		:= FALSE, 						(* Standard CAN Frame *)
									iByteCount			:= 8,							(* Number of bytes to send *)
									iData				:= TxData, 						(* Data frame *)
									oTransmitterId		=> ,
									oTooManyTransmitters=> , 
									oMsgSent			=> 
								);
							
					
								
	(*Info_To_AIM, ID=181*)
		(*TxData=16#00*)
			TxData[0]:=16#00;
			TxData[1]:=16#00;
			TxData[2]:=16#00;
			TxData[3]:=16#00;
			TxData[4]:=16#00;
			TxData[5]:=16#00;
			TxData[6]:=16#00;
			TxData[7]:=16#00;
		(*ASIGNACION DE LA VARIABLE A LA VARIABLE A ENVIAR (TxData)*)
		cl_split_dword( input := REAL_TO_WORD (AIM_TempMotor1_CAN),
									byte0=>TxData[0],
									byte1=>TxData[1],
								);
		cl_split_dword( input := REAL_TO_WORD (AIM_TempInverter1_CAN),
									byte0=>TxData[2],
									byte1=>TxData[3],
								);
		cl_split_dword( input := REAL_TO_WORD (AIM_TempMotor2_CAN),
									byte0=>TxData[4],
									byte1=>TxData[5],
								);
		cl_split_dword( input := REAL_TO_WORD (AIM_TempInverter2_CAN),
									byte0=>TxData[6],
									byte1=>TxData[7],
								);
					
									
				(*ENVÍO DE TxData*)
						FBTX_AIM_2(	iEnable				:= TRUE, 			(* Enables sending of messages *)
									iCAN				:= ADR(GVL.H_CAN_TX_6),			(* Structure for sending / receiving CAN messages *)
									iForceSend			:= FALSE,                       (* Force sending sends message immediately *)
									iTransmitRate		:= T#500MS, 						(* Cyclic transmission every 1000ms *)
									iCanId				:= 16#290,						(* CAN Id for message to send *)
									iCanIdExtended		:= FALSE, 						(* Standard CAN Frame *)
									iByteCount			:= 8,							(* Number of bytes to send *)
									iData				:= TxData, 						(* Data frame *)
									oTransmitterId		=> ,
									oTooManyTransmitters=> , 
									oMsgSent			=> 
								);
							
	(*Info_To_AIM, ID=182*)
		(*TxData=16#00*)
			TxData[0]:=16#00;
			TxData[1]:=16#00;
			TxData[2]:=16#00;
			TxData[3]:=16#00;
			TxData[4]:=16#00;
			TxData[5]:=16#00;
			TxData[6]:=16#00;
			TxData[7]:=16#00;
		(*ASIGNACION DE LA VARIABLE A LA VARIABLE A ENVIAR (TxData)*)
		cl_split_dword( input := REAL_TO_WORD (AIM_TempMotor3_CAN),
									byte0=>TxData[0],
									byte1=>TxData[1],
								);
		cl_split_dword( input := REAL_TO_WORD (AIM_TempInverter3_CAN),
									byte0=>TxData[2],
									byte1=>TxData[3],
								);
		cl_split_dword( input := REAL_TO_WORD (AIM_TempMotor4_CAN),
									byte0=>TxData[4],
									byte1=>TxData[5],
								);
		cl_split_dword( input := REAL_TO_WORD (AIM_TempInverter4_CAN),
									byte0=>TxData[6],
									byte1=>TxData[7],
								);
					
									
				(*ENVÍO DE TxData*)
						FBTX_AIM_3(	iEnable				:= TRUE, 			(* Enables sending of messages *)
									iCAN				:= ADR(GVL.H_CAN_TX_6),			(* Structure for sending / receiving CAN messages *)
									iForceSend			:= FALSE,                       (* Force sending sends message immediately *)
									iTransmitRate		:= T#500MS, 						(* Cyclic transmission every 100ms *)
									iCanId				:= 16#291,						(* CAN Id for message to send *)
									iCanIdExtended		:= FALSE, 						(* Standard CAN Frame *)
									iByteCount			:= 8,							(* Number of bytes to send *)
									iData				:= TxData, 						(* Data frame *)
									oTransmitterId		=> ,
									oTooManyTransmitters=> , 
									oMsgSent			=> 
								);
(*-----------------------------------------------FIN_AIM--------------------------------------------------------------*) 

*)

END_FUNCTION_BLOCK

